(* Logix 5000 project; controller Digital_Interlock_PLC vendor 1 type 14 code 196 rev 37.11; software revision 37.00 *)

TASK HeartbeatTask (periodic, rate 500 ms, priority 6, watchdog 10000 ms) : HeartbeatProgram
TASK MainTask (periodic, rate 5 ms, priority 5, watchdog 500 ms) : MainProgram
TASK ManageOptimizationTask (continuous, watchdog 500 ms) : ManageOptimizationProgram

MODULES
   Local : vendor 1 type 14 code 196 (5069 0, rev 37.11)
      PF1 : vendor 1 type 14 code 107 (Ethernet 10.10.10.48, rev 37.1)
      PR1 : vendor 887 type 12 code 42780 (Ethernet 10.10.10.6, rev 1.37, StandardDataDriven RPI 5 ms)
      ST1 : vendor 887 type 12 code 42780 (Ethernet 10.10.10.59, rev 1.37, StandardDataDriven RPI 5 ms)
END_MODULES

TYPE STR_MajorFault :
STRUCT
   LEN : DINT;
   DATA : SINT[300];
END_STRUCT
END_TYPE

TYPE UDT_Comms :
STRUCT
   PF : UDT_CommsHealth;
   PR : UDT_CommsHealth;
   ST : UDT_CommsHealth;
END_STRUCT
END_TYPE

TYPE UDT_CommsHealth :
STRUCT
   CommsError : BOOL;
   Healthy : BOOL;
   HeartbeatChanged : BOOL;
   Inhibited : BOOL;   // inhibited/uninhibited
   FaultInfo : DINT;
   Heartbeat : DINT;
   Inhibit : DINT;   // 0 to unihibit, 4 to inhibit.
   Instance : DINT;
   ArrivalPeriod_ms : REAL;
   Jitter_ms : REAL;
   LastArrivalPeriod_ms : REAL;
   Latency_ms : REAL;
   LatencyPeak_ms : REAL;
   LatencyAvg_ms : REAL;
   FaultCode : INT;   // 515 (disconnected during use), 516 (disconnected before controller run mode)
   Mode : INT;   // 0 (causes a major fault to be generated if any of the Module object connections fault while the controller is in Run mode) 2 (causes the Module object to enter Inhibited state after shutting down all the connections to the module.)
   Path : SINT[2];
END_STRUCT
END_TYPE

TYPE UDT_FaultRecord :
STRUCT
   TimeLow : DINT;
   TimeHigh : DINT;
   Type : INT;
   Code : INT;
   Info : DINT[11];
END_STRUCT
END_TYPE

TYPE UDT_FromLIC :   // Data that is exchanged with LIC Client
STRUCT
   EnableLineOptimization : BOOL;
   Deadband : DINT;
   FeedInterruptSetting : DINT;
   MaxCommandSpeed : DINT;
   MinCommandSpeed : DINT;
   Proportional : DINT;
   SampleRate : DINT;
   TargetFillPercentage : DINT;
   MachineList : STRING;
END_STRUCT
END_TYPE

TYPE UDT_MachineLFOProperties :   // UDT containing members needed for line flow optimization
STRUCT
   FeedInterruptStatus : BOOL;
   CommandedSpeed : DINT;
   CurrentSpeed : DINT;
   CurrentFillPercent : DINT;
   DeadBand : DINT;
   FeedInterruptSetting : DINT;
   PatternMaxSpeed : DINT;
   PatternMinSpeed : DINT;
   ReferenceSpeed : DINT;
   SpeedCalcRate : DINT;
   TargetFillPercent : DINT;
END_STRUCT
END_TYPE

TYPE UDT_MSG :
STRUCT
   To : DINT[33];
   From : DINT[33];
END_STRUCT
END_TYPE

TYPE UDT_ToLIC :
STRUCT
   FeedInterrupt : BOOL;   // Feed interrupt executed
   FeedInterrupted : BOOL;   // Interrupt completed
   CommsHealthy : BOOL;   // All machines are communicating
   MachinesConnected : BOOL[32];   // Boolean array that contains machine connection status
END_STRUCT
END_TYPE

ADD_ON_INSTRUCTION AOI_Calculate_Latency   (* revision 1.0 *)
VAR_INPUT
   Inp_DeviceHeartbeat : DINT; {required}
   Inp_CurrentTime_us : DINT; {required}
END_VAR
VAR_OUTPUT
   Out_LastTime_ms : DINT; {access Read Only, required}
   Out_HeartbeatChanged : BOOL; {access Read Only, required}
END_VAR
VAR
   CurrentTime_ms : DINT; {access None}
   PreviousTime_ms : DINT; {access None}
   PreviousHeartbeat : DINT; {access None}
   PreviousTime_us : DINT; {access None}
   dt_us : DINT; {access None}
   dt_ms : DINT; {access None}
END_VAR

ROUTINE Logic   (* structured text *)
   (*----------------------------------------------------------
   ROLLOVER-SAFE TIME DELTA
   	Inp_Timestamp_us is a microsecond counter that rolls to
   	zero each period. If the current timestamp is less than
   	the previous one, treat it as a rollover case.
   ----------------------------------------------------------*)
   
   if Inp_CurrentTime_us >= PreviousTime_us then
   	// Normal delta
       dt_us := Inp_CurrentTime_us - PreviousTime_us;
   else
   	// Rollover delta = remaining to modulus + current
   	dt_us := (1000000 - PreviousTime_us) + Inp_CurrentTime_us;
   end_if;
   
   // Convert microseconds to milliseconds for outputs.
   dt_ms := (dt_us) / 1000.0;
   
   
   if Inp_DeviceHeartbeat <> PreviousHeartbeat then
   	Out_HeartbeatChanged := 1;
   	Out_LastTime_ms := dt_ms - PreviousTime_ms;
   	PreviousTime_ms := dt_ms;
   else
   	Out_HeartbeatChanged := 0;
   end_if;
   
   PreviousHeartbeat := Inp_DeviceHeartbeat;
END_ROUTINE
END_ADD_ON_INSTRUCTION

ADD_ON_INSTRUCTION AOI_Detect_Heartbeat   (* revision 1.0 *)
VAR_INPUT
   Inp_Heartbeat : DINT; {required}
   Inp_WatchdogTime_ms : DINT; {visible}
END_VAR
VAR_OUTPUT
   Out_Heartbeat_Changed : BOOL; {access Read Only, visible}
   Out_WD_DN : BOOL; {access Read Only, visible}
   Out_WD_ACC : DINT; {access Read Only, visible}
   Out_WD_EN : BOOL; {access Read Only, visible}
   Out_Heartbeat_Healthy : BOOL; {access Read Only, required}
END_VAR
VAR
   PreviousHeartbeat : DINT; {access None}
   CurrentHeartbeat : DINT; {access None}
   HeartbeatWatchdog : FBD_TIMER; {access None}
END_VAR

ROUTINE Logic   (* structured text *)
   // Update current heartbeat value
   CurrentHeartbeat := Inp_Heartbeat;
   // Monitor changes in heartbeat
   Out_Heartbeat_Changed := (CurrentHeartbeat <> PreviousHeartbeat); //AND (NOT HeartbeatWatchdog.DN);
   
   // Check and set default preset for the watchdog if input preset is invalid (default to 10s)
   TONR(HeartbeatWatchdog);
   if Inp_WatchdogTime_ms <= 10000 then
   	HeartbeatWatchdog.PRE := 10000;
   else
   	HeartbeatWatchdog.PRE := Inp_WatchdogTime_ms;
   end_if;
   
   
   // Enable the watchdog timer if the heartbeat stops changing
   HeartbeatWatchdog.TimerEnable := NOT Out_Heartbeat_Changed;
   
   // Indicate bad health if the watchdog completes and no heartbeat change is detected
   Out_Heartbeat_Healthy := NOT (HeartbeatWatchdog.DN AND NOT Out_Heartbeat_Changed);
   
   // Reset the watchdog if both enabled and heartbeat changes detected
   if HeartbeatWatchdog.TimerEnable AND Out_Heartbeat_Changed then
       HeartbeatWatchdog.Reset := 1;
       HeartbeatWatchdog.TimerEnable := 0;
       HeartbeatWatchdog.Reset := 0;
   end_if;
   
   // Output the watchdog status flags
   Out_WD_DN := HeartbeatWatchdog.DN;
   Out_WD_ACC := HeartbeatWatchdog.ACC;
   Out_WD_EN := HeartbeatWatchdog.EN;
   
   // Store the current heartbeat for the next cycle
   PreviousHeartbeat := CurrentHeartbeat;
END_ROUTINE
END_ADD_ON_INSTRUCTION

ADD_ON_INSTRUCTION AOI_Monitor_Comms   (* revision 1.0 *)
// Latency-monitoring AOI tracks:
// Last heartbeat value
// Timestamp of last sample
// Latency (current, average, peak)
// Jitter (simple absolute-difference model)
VAR_INPUT
   Inp_Heartbeat : DINT; {required}   // heartbeat counter received from remote device
   Inp_Timestamp_us : DINT; {required}   // wall-clock microseconds from GSV(WallClockTime)
   Inp_MaxSameScans : DINT; {required}
   Inp_Rollover_us : DINT; {required}
   Inp_SmoothingFactor : REAL; {required}
   Inp_Reset : BOOL; {required}
END_VAR
VAR_OUTPUT
   Out_Latency_ms : REAL; {required}
   Out_LatencyAvg_ms : REAL; {access Read Only, required}
   Out_LatencyPeak_ms : REAL; {access Read Only, required}
   Out_Jitter_ms : REAL; {access Read Only, required}
   Out_Fresh : BOOL; {access Read Only, required}
   Out_HeartbeatOK : BOOL; {access Read Only, required}
END_VAR
VAR
   EMA : REAL; {access None}   // exponential smoothing accumulator
   FirstScan : BOOL; {access None}
   PreviousTime_us : DINT; {access None}
   PreviousHeartbeat : DINT; {access None}
   dt_us : DINT; {access None}
   dt_ms : REAL; {access None}
   SameValue : DINT; {access None}
   HeartbeatTimer : FBD_TIMER; {access None}
   EMA_prev : REAL; {access None}
   alpha : REAL; {access None}
   modulus : DINT; {access None}
END_VAR

ROUTINE Logic   (* structured text *)
// Latency-monitoring AOI
// It tracks:
// Last heartbeat value
// Timestamp of last sample
// Latency (current, average, peak)
// Jitter (simple absolute-difference model)
   (*
   |=================================================================|
   |						AOI_Comms_Monitor						  |
   |_________________________________________________________________|
   | Purpose:														  |
   | 	Measure time between successive remote heartbeats to estimate |
   |	comms latency, while handling microsecond timestamp rollover. |
   |																  |
   | Outputs are in milliseconds.									  |
   |_________________________________________________________________|
   *)
   
   (*--------------------------------------------------------------
   DISABLE / RESET BEHAVIOR
   	When disabled or reset, clear diagnostics and re-arm the
   	first-scan latch so the next enable reinitializes state.
   --------------------------------------------------------------*)
   
   if (NOT EnableIn) OR Inp_Reset then
   	FirstScan := 1;							// Force re-init on next enabled scan
   	PreviousTime_us := Inp_Timestamp_us;	// Seed previous timestamp to current
   	PreviousHeartbeat := Inp_Heartbeat;		// Seed previous heartbeat to current
   	EMA := 0;								// Clear exponential moving average accumulator
   	EMA_prev := 0;
   	SameValue := 0;
   
   	// Clear all status/diagnostics while disabled
   	Out_Fresh := 0;
   	Out_Latency_ms := 0;
   	Out_LatencyAvg_ms := 0;
   	Out_LatencyPeak_ms := 0;
   	Out_Jitter_ms := 0;
   	Out_HeartbeatOK := 0;
   end_if;
   
   (*--------------------------------------------------------------
   FIRST SAMPLE INITIALIZATION
   	On the first enabled scan, capture the baseline heartbeat
   	and timestamp so the next fresh value can compute a delta.
   --------------------------------------------------------------*)
   if FirstScan then
   	FirstScan := 0;							// Clear first-scan latch
   	PreviousHeartbeat := Inp_Heartbeat;		// Store current HB as baseline
   	PreviousTime_us := Inp_Timestamp_us;	// Store current timestamp as baseline
   
   	EMA := 0.0;								// Reset filter state
   	EMA_prev := 0.0;
   	SameValue := 0;
   
   	Out_HeartbeatOK := 1;					// Consider OK after initialization
   	Out_Fresh := 0;
   	Out_Latency_ms := 0.0;
   	Out_LatencyAvg_ms := 0.0;
   	Out_LatencyPeak_ms := 0.0;
   	Out_Jitter_ms := 0.0;
   end_if;
   
   
   (*--------------------------------------------------------------
   INPUT VALIDATION
   	Ensure smoothing factor is bounded between 0.0 and 1.0.
   	A heartbeat is considered "fresh" when its counter changes.
   --------------------------------------------------------------*)
   if Inp_SmoothingFactor < 0.0 then
   	Inp_SmoothingFactor := 0.0;
   end_if;
   
   if Inp_SmoothingFactor > 1.0 then
   	Inp_SmoothingFactor := 1.0;
   end_if;
   
   IF Inp_Rollover_us = 0 then
   	// Invalid modulus: mark unhealthy and bail (why: cannot compute deltas)
   	Out_Fresh := 0;
   	Out_HeartbeatOK := 0;
   end_if;
   
   
   (*--------------------------------------------------------------
   DETECT NEW HEARTBEAT
   	A heartbeat is considered "fresh" when its counter changes.
   --------------------------------------------------------------*)
   Out_Fresh := (Inp_Heartbeat <> PreviousHeartbeat);
   
   if Out_Fresh then
   	(*----------------------------------------------------------
   	ROLLOVER-SAFE TIME DELTA
   		Inp_Timestamp_us is a microsecond counter that rolls to
   		zero each period. If the current timestamp is less than
   		the previous one, treat it as a rollover case.
   	----------------------------------------------------------*)
   	if Inp_Timestamp_us >= PreviousTime_us then
   	    dt_us := Inp_Timestamp_us - PreviousTime_us;						// Normal delta
   	else
   		dt_us := (Inp_Rollover_us - PreviousTime_us) + Inp_Timestamp_us;	// Rollover delta = remaining to modulus + current
   	end_if;
   
   	dt_ms := (dt_us) / 1000.0;			// Convert microseconds to milliseconds for outputs.
   
   	Out_Latency_ms := dt_ms;			// Latency for this heartbeat interval
   
   	if dt_ms > Out_LatencyPeak_ms then
   		Out_LatencyPeak_ms := dt_ms;	// Track worst-case latency
   	end_if;
   
   	(*----------------------------------------------------------
   	SMOOTHED AVERAGE (EMA)
   		EMA is a low-pass filter:
   			EMA := (1 - alpha) * EMA + alpha * sample
   		Here, alpha is provided as Inp_SmoothingFactor.
   	----------------------------------------------------------*)
   
   	EMA := (1-Inp_SmoothingFactor) * EMA + Inp_SmoothingFactor * dt_ms;
   
   	Out_LatencyAvg_ms := EMA;
   
   	(*----------------------------------------------------------
   	JITTER ESTIMATE
   		Jitter is modeled as the absolute deviation of the
   		latest sample from the smoothed average.
   	----------------------------------------------------------*)
   	Out_Jitter_ms := ABS(dt_ms - EMA);
   
   	(*----------------------------------------------------------
   	UPDATE HISTORY
   		Persist current values for the next fresh heartbeat
   		comparison and mark comms as healthy.
   	----------------------------------------------------------*)
   	PreviousHeartbeat := Inp_Heartbeat;
   	PreviousTime_us := Inp_Timestamp_us;
   	SameValue := 0;
   	Out_HeartbeatOK := 1;
   
   else
   	// Heartbeat did not change this scan; track consecutive repeats
   	if SameValue < Inp_MaxSameScans then
   		SameValue := SameValue + 1;
   	end_if;
   
   	// After N identical scans, consider comms unhealthy
   	if (SameValue >= Inp_MaxSameScans) then
   		Out_HeartbeatOK := 0;
   	end_if;
   end_if;
END_ROUTINE
END_ADD_ON_INSTRUCTION

ADD_ON_INSTRUCTION AOI_Optimize_Flow   (* revision 1.0 *)
// Line Speed Adjustment
VAR_INPUT
   Inp_CurrentSpeed : DINT; {required}   // Current speed of the target machine (KPM)
   Inp_ReferenceSpeed : DINT; {required}   // Reference speed of the downstream machine (KPM)
   Inp_CurrentFillPercent : DINT; {required}
   Inp_TargetFillPercent : DINT; {required}   // Target Fill Percentage, the desired fill percentage to achieve by adjusting speeds (%)
   Inp_MaxSpeed : DINT; {required}   // Maximum speed of job (KPM)
   Inp_MinSpeed : DINT; {required}   // Minimum speed of target machine (KPM)
   Inp_FeedInterruptSetting : DINT; {required}   // Value set by LIC Client user interface
   Inp_SpeedCalcRate : DINT; {required}   // Rate of speed calculations
END_VAR
VAR_OUTPUT
   Out_CommandSpeed : DINT; {required}
   Out_FeedInterrupt : BOOL; {required}   // Value set to TRUE, when the Reference Fill % is equal to or greater than the Feed Interrupt Setting LIC Client user input).
END_VAR
VAR
   SpeedCalcTimer : TIMER;
   ProportionalGain : DINT;   // Proportial multiple to adjust aggressiveness of changes to speed commands, limited to [0.5 - 1.2]
   DeadBand : DINT;   // Value that represents the amount of percentage points from target fill percentage that the current fill percentage must be before calculating command speed
   LowerDeadBand : DINT;
   UpperDeadBand : DINT;
END_VAR

ROUTINE Logic   (* ladder *)
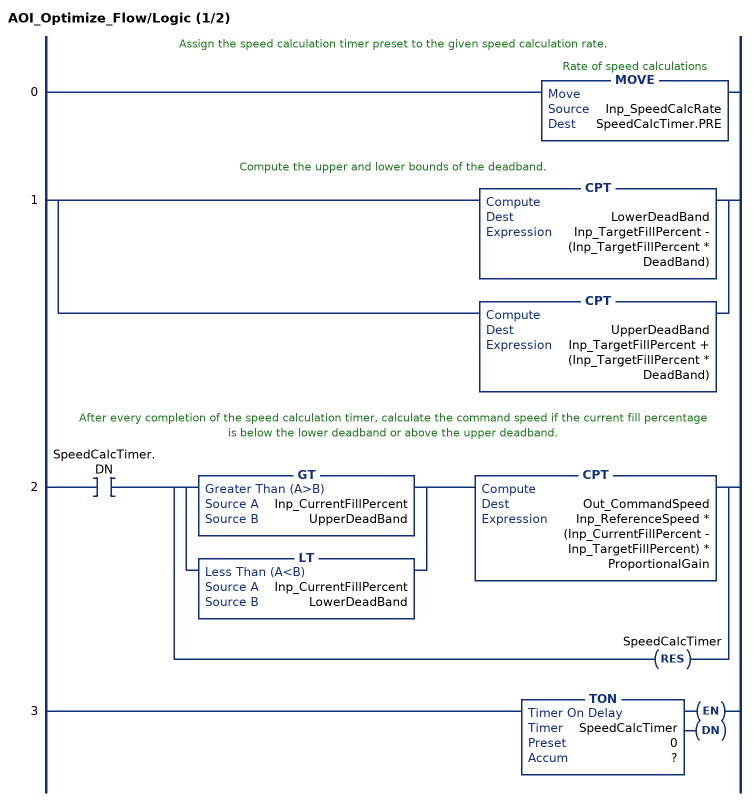
   // Assign the speed calculation timer preset to the given speed calculation rate.
   0: MOVE(Inp_SpeedCalcRate,SpeedCalcTimer.PRE);
   // Compute the upper and lower bounds of the deadband.
   1: [CPT(LowerDeadBand,Inp_TargetFillPercent - (Inp_TargetFillPercent * DeadBand)) ,CPT(UpperDeadBand,Inp_TargetFillPercent + (Inp_TargetFillPercent * DeadBand)) ];
   // After every completion of the speed calculation timer, calculate the command speed if the current fill percentage is below the lower deadband or above the upper deadband.
   2: XIC(SpeedCalcTimer.DN)[[GT(Inp_CurrentFillPercent,UpperDeadBand) ,LT(Inp_CurrentFillPercent,LowerDeadBand) ] CPT(Out_CommandSpeed,Inp_ReferenceSpeed * (Inp_CurrentFillPercent - Inp_TargetFillPercent) * ProportionalGain) ,RES(SpeedCalcTimer) ];
   3: TON(SpeedCalcTimer,?,?);
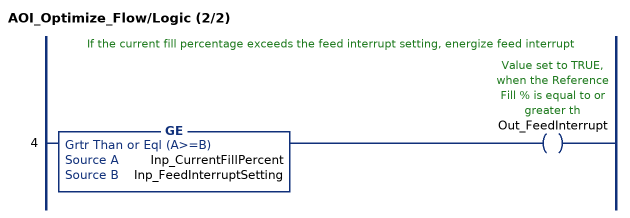
   // If the current fill percentage exceeds the feed interrupt setting, energize feed interrupt
   4: GE(Inp_CurrentFillPercent,Inp_FeedInterruptSetting)OTE(Out_FeedInterrupt);
END_ROUTINE
END_ADD_ON_INSTRUCTION

VAR_GLOBAL   (* controller tags *)
   _DEBUG : BOOL;
   AlwaysTrue : BOOL := 1; {constant}
   CommsStatus : DINT := 7;
        .0   // Bit for PREFEEDER Comms Status
        .3   // Bit for LIC Comms Status
        .2   // Bit for STACKER Comms Status
        .1   // Bit for PRESS Comms Status
   CurrentTime : DINT[7] := ([0] := 2026, [1] := 2, [2] := 23, [3] := 14, [4] := 10, [5] := 41, [6] := 704831);
   EnableLineOptimization : BOOL;
   FromPrefeeder : DINT[33] := ([0] := 264, [3] := 734);   // DINTs used: 0-2
        [0].8   // (Pre-Feeder -> Press) FromPrefeeder.MachineOpenCloseDisable
        [0].11   // (Pre-Feeder -> Press) FromPrefeeder.ReadyToRaise
        [0].1   // (Pre-Feeder -> Press) FromPrefeeder.AuxTamperAirLeft
        [0].10   // (Pre-Feeder -> Press) FromPrefeeder.ReadyForSetup
        [0].7   // (Pre-Feeder -> Press) FromPrefeeder.FeedBoardOk
        [2]   // (Pre-Feeder -> Press) FromPrefeeder.PatternMaxSpeed
        [0].5   // (Pre-Feeder -> Press) FromPrefeeder.EstopFeedbackChannel1
        [0].6   // (Pre-Feeder -> Press) FromPrefeeder.EstopFeedbackChannel2
        [0].2   // (Pre-Feeder -> Press) FromPrefeeder.BackstopInhibit
        [0].4   // (Pre-Feeder -> Press) FromPrefeeder.ExtendoUpDown
        [0].18   // Spare
        [4]   // (Pre-Feeder -> Press) FromPrefeeder.Spare1
        [1]   // (Pre-Feeder -> Press) FromPrefeeder.CurrentSpeed
        [3]   // (Pre-Feeder -> Press) FromPrefeeder.Heartbeat
        [5]   // (Pre-Feeder -> Press) FromPrefeeder.Spare2
        [0].19   // Spare
        [0].20   // Spare
        [0].12   // (Pre-Feeder -> Press) FromPrefeeder.RunEmpty
        [0].21   // Spare
        [0].22   // Spare
        [0].23   // Spare
        [0].24   // Spare
        [0]   // Bits used: 0-17
        [0].9   // (Pre-Feeder -> Press) FromPrefeeder.OpenMachineOk
        [0].16   // (Pre-Feeder -> Press) FromPrefeeder.Empty
        [0].17   // (Pre-Feeder -> Press) FromPrefeeder.Spare
        [0].0   // (Pre-Feeder -> Press) FromPrefeeder.AuxTamperAirRight
        [10]   // Spare
        [11]   // Spare
        [12]   // Spare
        [13]   // Spare
        [14]   // Spare
        [15]   // Spare
        [16]   // Spare
        [17]   // Spare
        [18]   // Spare
        [19]   // Spare
        [20]   // Spare
        [21]   // Spare
        [22]   // Spare
        [23]   // Spare
        [24]   // Spare
        [25]   // Spare
        [26]   // Spare
        [27]   // Spare
        [28]   // Spare
        [0].13   // (Pre-Feeder -> Floor Conv) FromPrefeeder.RunForward
        [0].14   // (Pre-Feeder -> Floor Conv) FromPrefeeder.RunReverse
        [0].15   // (Pre-Feeder -> Press) FromPrefeeder.TamperInterrupt
        [0].3   // (Pre-Feeder -> Floor Conv) FromPrefeeder.CallForStack
        [0].25   // Spare
        [0].26   // Spare
        [0].27   // Spare
        [0].28   // Spare
        [0].29   // Spare
        [0].30   // Spare
        [0].31   // Spare
        [29]   // Spare
        [30]   // Spare
        [31]   // Spare
        [32]   // Spare
        [6]   // Spare
        [7]   // Spare
        [8]   // Spare
        [9]   // Spare
   FromPrefeeder_Copied : REAL[20];
   FromPress : DINT[33] := ([0] := 60635, [1] := 125, [2] := 75, [3] := 16, [4] := 888, [5] := 1143336141, [7] := 1153686979, [8] := 1153638072, [9] := 1153709834, [14] := 1146431734, [15] := -1098572104);
   FromPress_Copied : REAL[20];
   FromStacker : DINT[33];   // DINTS used: 0-22
        [4].7   // (Stacker -> Press) fromStacker.DieCutter.blnRegisterStopAdjustRq
        [4].3   // (Stacker -> Press) fromStacker.FeedInterruptStatus
        [4].6   // (Stacker -> Press) fromStacker.DieCutter.blnRegisterAdjustRq
        [4].9   // (Stacker -> Press) fromStacker.DieCutter.blnSidewaysStopAdjustRq
        [5].0   // (Stacker -> Press) fromStacker.PrintStation[7].blnRegisterStopAdjustRq
        [4].4   // (Stacker -> Press) fromStacker.DieCutter.blnFast
        [10]   // (Stacker -> Press) fromStacker.PrintStation[3].fltDesiredRegisterAdjust
        [4].26   // (Stacker -> Press) fromStacker.PrintStation[1].blnRegisterStopAdjustRq
        [4].8   // (Stacker -> Press) fromStacker.DieCutter.blnSidewaysAdjustRq
        [7]   // (Stacker -> Press) fromStacker.DieCutter.fltDesiredRegisterAdjust
        [15]   // (Stacker -> Press) fromStacker.DieCutter.fltDesiredSidewaysAdjust
        [4].10   // (Stacker -> Press) fromStacker.DieCutter.blnSpeedChangeRq
        [5].1   // (Stacker -> Press) fromStacker.PrintStation[1].blnSidewaysStopAdjustRq
        [4].12   // (Stacker -> Press) fromStacker.PrintStation[1].blnRegisterAdjustRq
        [5].2   // (Stacker -> Press) fromStacker.PrintStation[2].blnSidewaysStopAdjustRq
        [4].11   // (Stacker -> Press) fromStacker.DieCutter.blnSpeedChangeStopRq
        [5].3   // (Stacker -> Press) fromStacker.PrintStation[3].blnSidewaysStopAdjustRq
        [11]   // (Stacker -> Press) fromStacker.PrintStation[4].fltDesiredRegisterAdjust
        [8]   // (Stacker -> Press) fromStacker.PrintStation[1].fltDesiredRegisterAdjust
        [5].4   // (Stacker -> Press) fromStacker.PrintStation[4].blnSidewaysStopAdjustRq
        [9]   // (Stacker -> Press) fromStacker.PrintStation[2].fltDesiredRegisterAdjust
        [5].5   // (Stacker -> Press) fromStacker.PrintStation[5].blnSidewaysStopAdjustRq
        [4].13   // (Stacker -> Press) fromStacker.PrintStation[2].blnRegisterAdjustRq
        [5].6   // (Stacker -> Press) fromStacker.PrintStation[6].blnSidewaysStopAdjustRq
        [6]   // (Stacker -> Press) fromStacker.DieCutter.uiDesiredSpeedKpm
        [4].14   // (Stacker -> Press) fromStacker.PrintStation[3].blnRegisterAdjustRq
        [4].15   // (Stacker -> Press) fromStacker.PrintStation[4].blnRegisterAdjustRq
        [4].16   // (Stacker -> Press) fromStacker.PrintStation[5].blnRegisterAdjustRq
        [12]   // (Stacker -> Press) fromStacker.PrintStation[5].fltDesiredRegisterAdjust
        [13]   // (Stacker -> Press) fromStacker.PrintStation[6].fltDesiredRegisterAdjust
        [14]   // (Stacker -> Press) fromStacker.PrintStation[7].fltDesiredRegisterAdjust
        [16]   // (Stacker -> Press) fromStacker.PrintStation[1].fltDesiredSidewaysAdjust
        [17]   // (Stacker -> Press) fromStacker.PrintStation[2].fltDesiredSidewaysAdjust
        [18]   // (Stacker -> Press) fromStacker.PrintStation[3].fltDesiredSidewaysAdjust
        [19]   // (Stacker -> Press) fromStacker.PrintStation[4].fltDesiredSidewaysAdjust
        [20]   // (Stacker -> Press) fromStacker.PrintStation[5].fltDesiredSidewaysAdjust
        [21]   // (Stacker -> Press) fromStacker.PrintStation[6].fltDesiredSidewaysAdjust
        [22]   // (Stacker -> Press) fromStacker.PrintStation[7].fltDesiredSidewaysAdjust
        [5].7   // (Stacker -> Press) fromStacker.PrintStation[7].blnSidewaysStopAdjustRq
        [4].27   // (Stacker -> Press) fromStacker.PrintStation[2].blnRegisterStopAdjustRq
        [4].17   // (Stacker -> Press) fromStacker.PrintStation[6].blnRegisterAdjustRq
        [4].28   // (Stacker -> Press) fromStacker.PrintStation[3].blnRegisterStopAdjustRq
        [4].18   // (Stacker -> Press) fromStacker.PrintStation[7].blnRegisterAdjustRq
        [4].19   // (Stacker -> Press) fromStacker.PrintStation[1].blnSidewaysAdjustRq
        [4].5   // (Stacker -> Press) fromStacker.DieCutter.blnSlow
        [4].2   // (Stacker -> Press) fromStacker.RolledOutStatus
        [4].0   // (Stacker -> Press) fromStacker.RunPermissive
        [4].29   // (Stacker -> Press) fromStacker.PrintStation[4].blnRegisterStopAdjustRq
        [4].30   // (Stacker -> Press) fromStacker.PrintStation[5].blnRegisterStopAdjustRq
        [4].31   // (Stacker -> Press) fromStacker.PrintStation[6].blnRegisterStopAdjustRq
        [4].20   // (Stacker -> Press) fromStacker.PrintStation[2].blnSidewaysAdjustRq
        [4].21   // (Stacker -> Press) fromStacker.PrintStation[3].blnSidewaysAdjustRq
        [2]   // (Stacker -> Press) fromStacker.PatternMaxSpeed
        [4].1   // (Stacker -> Press) fromStacker.FeedRestart
        [0]   // (Stacker -> Press) fromStacker.Heartbeat
        [3]   // (Stacker -> Press) fromStacker.FillPercentage
        [5]   // Bits used: 0-7
        [1]   // (Stacker -> Press) fromStacker.CurrentSpeed
        [4].22   // (Stacker -> Press) fromStacker.PrintStation[4].blnSidewaysAdjustRq
        [4]   // Bits used: 0-31
        [4].23   // (Stacker -> Press) fromStacker.PrintStation[5].blnSidewaysAdjustRq
        [4].24   // (Stacker -> Press) fromStacker.PrintStation[6].blnSidewaysAdjustRq
        [4].25   // (Stacker -> Press) fromStacker.PrintStation[7].blnSidewaysAdjustRq
        [23]   // Spare
        [24]   // Spare
        [25]   // Spare
        [26]   // Spare
        [27]   // Spare
        [28]   // Spare
        [29]   // Spare
        [30]   // Spare
        [31]   // Spare
        [32]   // Spare
   FromStacker_Copied : REAL[20];
   HeartbeatCounter : INT := 832;
   PF_Comms : UDT_CommsHealth;
        .CommsError   // Prefeeder comms error
   PR_Comms : UDT_CommsHealth;
        .CommsError   // Press comms error
   PrefeederData : UDT_MSG := (To[8] := 727, To[9] := 7, From[0] := 264, From[3] := 727);
   PrefeederLFO : UDT_MachineLFOProperties;
   PrefeederLFO_AOI : AOI_Optimize_Flow;
   PrefeederMSG : MESSAGE;
        MessageParameters(ServiceCode := 16#004d, LocalElement := PrefeederData.To[0], ...)
   PressLatency_AOI : AOI_Calculate_Latency;
   PressLFO : UDT_MachineLFOProperties;
   PressLFO_AOI : AOI_Optimize_Flow;
   ST_Comms : UDT_CommsHealth;
        .CommsError   // Stacker comms error
   StackerLFO : UDT_MachineLFOProperties;
   StackerLFO_AOI : AOI_Optimize_Flow;
   ToPrefeeder2 : DINT[33];   // DINTs used: 0-11
        [4]   // (Press -> Pre-Feeder) ToPrefeeder.HopperHeightSetpoint
        [0].10   // ToPrefeeder.ShuttleCarAtPrefeeder (Floor Conv -> Prefeeder)
        [0].9   // ToPrefeeder.StackReadyInFeed (Floor Conv -> Prefeeder)
        [0].4   // ToPrefeeder.LastStack (Floor Conv -> Prefeeder)
        [7]   // (Press -> Pre-Feeder) ToPrefeeder.LinearSpeedActual
        [0].3   // ToPrefeeder.ExtendoFollowBackstopDown (Press -> Pre-Feeder)
        [0].2   // ToPrefeeder.ExtendoFollowBackstopUp (Press -> Pre-Feeder)
        [0].8   // ToPrefeeder.RequestOpen (Press -> Pre-Feeder)
        [5]   // (Press -> Pre-Feeder) ToPrefeeder.HopperHeightMin
        [9]   // (Interlock -> Pre-Feeder) ToPrefeeder.CommsStatus
        [27]   // Spare
        [28]   // Spare
        [29]   // Spare
        [30]   // Spare
        [0].25   // Spare
        [0].6   // ToPrefeeder.MachineInFeedMode (Press -> Pre-Feeder)
        [0].26   // Spare
        [0].27   // Spare
        [31]   // Spare
        [0].28   // Spare
        [0].29   // Spare
        [0].30   // Spare
        [0].31   // Spare
        [0].7   // ToPrefeeder.MachineRunning (Press -> Pre-Feeder)
        [0].5   // ToPrefeeder.LoadHopper (Press -> Pre-Feeder)
        [1]   // (Press -> Pre-Feeder) ToPrefeeder.CommandedSpeed
        [2]   // (Press -> Pre-Feeder) ToPrefeeder.BoardCaliper
        [8]   // Prefeeder[8] (ToPrefeeder.Heartbeat)
        [10]   // (Press -> Pre-Feeder) ToPrefeeder.Spare1
        [11]   // (Press -> Pre-Feeder) ToPrefeeder.Spare2
        [0].1   // ToPrefeeder.ConvRunning (Floor Conv -> Prefeeder)
        [0]   // Bits used: 0-10
        [0].0   // ToPrefeeder.ClosedLocked (Press -> Pre-Feeder)
        [3]   // (Press -> Pre-Feeder) ToPrefeeder.FeedHopperHeight
        [6]   // (Press -> Pre-Feeder) ToPrefeeder.LinearSpeedSetpoint
        [0].11   // Spare
        [0].12   // Spare
        [0].13   // Spare
        [0].14   // Spare
        [0].15   // Spare
        [0].16   // Spare
        [0].17   // Spare
        [12]   // Spare
        [13]   // Spare
        [14]   // Spare
        [15]   // Spare
        [16]   // Spare
        [17]   // Spare
        [18]   // Spare
        [19]   // Spare
        [20]   // Spare
        [21]   // Spare
        [22]   // Spare
        [23]   // Spare
        [24]   // Spare
        [25]   // Spare
        [26]   // Spare
        [0].18   // Spare
        [0].19   // Spare
        [0].20   // Spare
        [0].21   // Spare
        [0].22   // Spare
        [0].23   // Spare
        [0].24   // Spare
   ToPress : DINT[40];   // DINTs used: 0-32
        [10].6   // (Stacker -> Press) fromStacker.DieCutter.blnRegisterAdjustRq
        [10].8   // (Stacker -> Press) fromStacker.DieCutter.blnSidewaysAdjustRq
        [0].1   // (Pre-Feeder -> Press) FromPrefeeder.AuxTamperAirLeft
        [12]   // (Stacker -> Press) fromStacker.DieCutter.uiDesiredSpeedKpm
        [0].11   // (Pre-Feeder -> Press) FromPrefeeder.ReadyToRaise
        [0].5   // (Pre-Feeder -> Press) FromPrefeeder.EstopFeedbackChannel1
        [0].10   // (Pre-Feeder -> Press) FromPrefeeder.ReadyForSetup
        [10].11   // (Stacker -> Press) fromStacker.DieCutter.blnSpeedChangeStopRq
        [10].26   // (Stacker -> Press) fromStacker.PrintStation[1].blnRegisterStopAdjustRq
        [10].7   // (Stacker -> Press) fromStacker.DieCutter.blnRegisterStopAdjustRq
        [10].9   // (Stacker -> Press) fromStacker.DieCutter.blnSidewaysStopAdjustRq
        [10].27   // (Stacker -> Press) fromStacker.PrintStation[2].blnRegisterStopAdjustRq
        [10].28   // (Stacker -> Press) fromStacker.PrintStation[3].blnRegisterStopAdjustRq
        [0].17   // (Pre-Feeder -> Press) FromPrefeeder.FeedInterrupt
        [10].4   // (Stacker -> Press) fromStacker.DieCutter.blnFast
        [10].29   // (Stacker -> Press) fromStacker.PrintStation[4].blnRegisterStopAdjustRq
        [10].3   // (Stacker -> Press) FromStacker.FeedInterruptStatus
        [10].10   // (Stacker -> Press) fromStacker.DieCutter.blnSpeedChangeRq
        [32].0   // (Interlock -> Prefeeder) FromInterlock.PrefeederCommsStatus
        [10].5   // (Stacker -> Press) fromStacker.DieCutter.blnSlow
        [10].30   // (Stacker -> Press) fromStacker.PrintStation[5].blnRegisterStopAdjustRq
        [10].31   // (Stacker -> Press) fromStacker.PrintStation[6].blnRegisterStopAdjustRq
        [0].8   // (Pre-Feeder -> Press) FromPrefeeder.MachineOpenCloseDisable
        [0].6   // (Pre-Feeder -> Press) FromPrefeeder.EstopFeedbackChannel2
        [13]   // (Stacker -> Press) fromStacker.DieCutter.fltDesiredRegisterAdjust
        [21]   // (Stacker -> Press) fromStacker.DieCutter.fltDesiredSidewaysAdjust
        [0].2   // (Pre-Feeder -> Press) FromPrefeeder.BackstopInhibit
        [0].7   // (Pre-Feeder -> Press) FromPrefeeder.FeedBoardOk
        [2]   // (Pre-Feeder -> Press) FromPrefeeder.PatternMaxSpeed
        [31]   // (Interlock -> Press) FromInterlock.CommandedSpeed
        [14]   // (Stacker -> Press) fromStacker.PrintStation[1].fltDesiredRegisterAdjust
        [15]   // (Stacker -> Press) fromStacker.PrintStation[2].fltDesiredRegisterAdjust
        [32].2   // (Interlock -> Stacker) FromInterlock.StackerCommsStatus
        [16]   // (Stacker -> Press) fromStacker.PrintStation[3].fltDesiredRegisterAdjust
        [10].12   // (Stacker -> Press) fromStacker.PrintStation[1].blnRegisterAdjustRq
        [0].0   // (Pre-Feeder -> Press) FromPrefeeder.AuxTamperAirRight
        [17]   // (Stacker -> Press) fromStacker.PrintStation[4].fltDesiredRegisterAdjust
        [18]   // (Stacker -> Press) fromStacker.PrintStation[5].fltDesiredRegisterAdjust
        [10].13   // (Stacker -> Press) fromStacker.PrintStation[2].blnRegisterAdjustRq
        [19]   // (Stacker -> Press) fromStacker.PrintStation[6].fltDesiredRegisterAdjust
        [11].0   // (Stacker -> Press) fromStacker.PrintStation[7].blnRegisterStopAdjustRq
        [20]   // (Stacker -> Press) fromStacker.PrintStation[7].fltDesiredRegisterAdjust
        [22]   // (Stacker -> Press) fromStacker.PrintStation[1].fltDesiredSidewaysAdjust
        [0].4   // (Pre-Feeder -> Press) FromPrefeeder.ExtendoUpDown
        [10].14   // (Stacker -> Press) fromStacker.PrintStation[3].blnRegisterAdjustRq
        [4]   // (Pre-Feeder -> Press) FromPrefeeder.Spare1
        [0].9   // (Pre-Feeder -> Press) FromPrefeeder.OpenMachineOk
        [5]   // (Pre-Feeder -> Press) FromPrefeeder.Spare2
        [11].1   // (Stacker -> Press) fromStacker.PrintStation[1].blnSidewaysStopAdjustRq
        [10].2   // (Stacker -> Press) FromStacker.RolledOutStatus
        [11].2   // (Stacker -> Press) fromStacker.PrintStation[2].blnSidewaysStopAdjustRq
        [11].3   // (Stacker -> Press) fromStacker.PrintStation[3].blnSidewaysStopAdjustRq
        [0].12   // (Pre-Feeder -> Press) FromPrefeeder.RunEmpty
        [32].3   // Spare
        [0].16   // (Pre-Feeder -> Press) FromPrefeeder.Empty
        [32].4   // Spare
        [32].5   // Spare
        [10].1   // (Stacker -> Press) FromStacker.FeedRestart
        [11]   // Bits used: 0-7
        [3]   // (Pre-Feeder -> Press) FromPrefeeder.Heartbeat
        [10]   // Bits uses: 0-31
        [32].6   // Spare
        [32].7   // Spare
        [32].8   // Spare
        [32].9   // Spare
        [32].10   // Spare
        [32]   // Bits used: 0-2
        [32].11   // Spare
        [9]   // (Stacker -> Press) FromStacker.FillPercentage
        [1]   // (Pre-Feeder -> Press) FromPrefeeder.CurrentSpeed
        [10].15   // (Stacker -> Press) fromStacker.PrintStation[4].blnRegisterAdjustRq
        [10].0   // (Stacker -> Press) FromStacker.RunPermissive
        [7]   // (Stacker -> Press) FromStacker.CurrentSpeed
        [11].4   // (Stacker -> Press) fromStacker.PrintStation[4].blnSidewaysStopAdjustRq
        [8]   // (Stacker -> Press) FromStacker.PatternMaxSpeed
        [11].5   // (Stacker -> Press) fromStacker.PrintStation[5].blnSidewaysStopAdjustRq
        [32].12   // Spare
        [29]   // (Stacker -> Press) fromStacker.Spare1
        [10].16   // (Stacker -> Press) fromStacker.PrintStation[5].blnRegisterAdjustRq
        [30]   // (Stacker -> Press) fromStacker.Spare2
        [6]   // (Stacker -> Press) FromStacker.Heartbeat
        [11].6   // (Stacker -> Press) fromStacker.PrintStation[6].blnSidewaysStopAdjustRq
        [0]   // Bits used: 0-18
        [0].13   // (Pre-Feeder -> Floor Conv) FromPrefeeder.RunForward
        [0].14   // (Pre-Feeder -> Floor Conv) FromPrefeeder.RunReverse
        [0].15   // (Pre-Feeder -> Press) FromPrefeeder.TamperInterrupt
        [0].3   // (Pre-Feeder -> Floor Conv) FromPrefeeder.CallForStack
        [32].1   // (Interlock -> Press) FromInterlock.PressCommsStatus
        [0].18   // (Pre-Feeder -> Press) FromPrefeeder.Spare
        [10].17   // (Stacker -> Press) fromStacker.PrintStation[6].blnRegisterAdjustRq
        [10].18   // (Stacker -> Press) fromStacker.PrintStation[7].blnRegisterAdjustRq
        [10].19   // (Stacker -> Press) fromStacker.PrintStation[1].blnSidewaysAdjustRq
        [10].20   // (Stacker -> Press) fromStacker.PrintStation[2].blnSidewaysAdjustRq
        [10].21   // (Stacker -> Press) fromStacker.PrintStation[3].blnSidewaysAdjustRq
        [10].22   // (Stacker -> Press) fromStacker.PrintStation[4].blnSidewaysAdjustRq
        [10].23   // (Stacker -> Press) fromStacker.PrintStation[5].blnSidewaysAdjustRq
        [10].24   // (Stacker -> Press) fromStacker.PrintStation[6].blnSidewaysAdjustRq
        [10].25   // (Stacker -> Press) fromStacker.PrintStation[7].blnSidewaysAdjustRq
        [11].7   // (Stacker -> Press) fromStacker.PrintStation[7].blnSidewaysStopAdjustRq
        [23]   // (Stacker -> Press) fromStacker.PrintStation[2].fltDesiredSidewaysAdjust
        [24]   // (Stacker -> Press) fromStacker.PrintStation[3].fltDesiredSidewaysAdjust
        [25]   // (Stacker -> Press) fromStacker.PrintStation[4].fltDesiredSidewaysAdjust
        [26]   // (Stacker -> Press) fromStacker.PrintStation[5].fltDesiredSidewaysAdjust
        [27]   // (Stacker -> Press) fromStacker.PrintStation[6].fltDesiredSidewaysAdjust
        [28]   // (Stacker -> Press) fromStacker.PrintStation[7].fltDesiredSidewaysAdjust
        [32].13   // Spare
        [32].14   // Spare
        [32].15   // Spare
        [32].16   // Spare
        [32].17   // Spare
        [32].18   // Spare
        [32].19   // Spare
        [32].20   // Spare
        [32].21   // Spare
        [32].22   // Spare
        [32].23   // Spare
        [32].24   // Spare
        [32].25   // Spare
        [32].26   // Spare
        [32].27   // Spare
        [32].28   // Spare
        [32].29   // Spare
        [32].30   // Spare
        [32].31   // Spare
   ToStacker : DINT[33] := ([0] := 60635, [1] := 125, [2] := 75, [3] := 16, [4] := 888, [5] := 1143336141, [7] := 1153686979, [8] := 1153638072, [9] := 1153709834, [14] := 1146431734, [15] := -1098572104);   // DINTS used: 0-23
        [3].15   // (Press -> Stacker) toStacker.PrintStation[1].blnSideWaysActive
        [3].16   // (Press -> Stacker) toStacker.PrintStation[2].blnSideWaysActive
        [3].22   // (LIC -> Stacker) toStacker.DownstreamReady(StraightThru)
        [3].5   // (Press -> Stacker) toStacker.DieCutter.blnRegistrationActive
        [3].8   // (Press -> Stacker) toStacker.PrintStation[1].blnRegistrationActive
        [5]   // (Press -> Stacker) toStacker.DieCutter.fltActualRegisterPosition
        [3].9   // (Press -> Stacker) toStacker.PrintStation[2].blnRegistrationActive
        [3].6   // (Press -> Stacker) toStacker.DieCutter.blnSidewaysAcitve
        [6]   // (Press -> Stacker) toStacker.DieCutter.fltActualSidewaysPosition
        [7]   // (Press -> Stacker) toStacker.PrintStation[1].fltActualRegisterPosition
        [3].17   // (Press -> Stacker) toStacker.PrintStation[3].blnSideWaysActive
        [8]   // (Press -> Stacker) toStacker.PrintStation[2].fltActualRegisterPosition
        [3].25   // (Press -> Stacker) toStacker.DieCutter.blnDieDrumReferenced
        [3].18   // (Press -> Stacker) toStacker.PrintStation[4].blnSideWaysActive
        [9]   // (Press -> Stacker) toStacker.PrintStation[3].fltActualRegisterPosition
        [3].19   // (Press -> Stacker) toStacker.PrintStation[5].blnSideWaysActive
        [3].20   // (Press -> Stacker) toStacker.PrintStation[6].blnSideWaysActive
        [3].21   // (Press -> Stacker) toStacker.PrintStation[7].blnSideWaysActive
        [3].4   // (Press -> Stacker) toStacker.SheetCountPulseStatus
        [3].7   // (Press -> Stacker) toStacker.DieCutter.blnSpeedChangeActive
        [22]   // (Press -> Stacker) toStacker.Spare1
        [23]   // (Press -> Stacker) toStacker.Spare2
        [3].23   // (LIC -> Stacker) toStacker.ReadyRightAngleForward
        [3].24   // (LIC -> Stacker) toStacker.ReadyRightAngleReverse
        [4]   // (Press -> Stacker) toStacker.DieCutter.uiActualSpeedKpm
        [24]   // Spare
        [25]   // Spare
        [3].0   // (Press -> Stacker) toStacker.RollInPermissive
        [26]   // Spare
        [27]   // Spare
        [28]   // Spare
        [29]   // Spare
        [30]   // Spare
        [31]   // Spare
        [3].2   // (Press -> Stacker) toStacker.VOSReset
        [3].3   // (Press -> Stacker) toStacker.VOSStart
        [21]   // (Interlock -> Stacker) toStacker.CommsStatus
        [1]   // (Press -> Stacker) toStacker.CommandedSpeed
        [0]   // (Press -> Stacker) toStacker.Heartbeat
        [2]   // (Press -> Stacker) toStacker.PressCurrentSpeed
        [3].1   // (Press -> Stacker) toStacker.RunPermissive
        [10]   // (Press -> Stacker) toStacker.PrintStation[4].fltActualRegisterPosition
        [11]   // (Press -> Stacker) toStacker.PrintStation[5].fltActualRegisterPosition
        [12]   // (Press -> Stacker) toStacker.PrintStation[6].fltActualRegisterPosition
        [13]   // (Press -> Stacker) toStacker.PrintStation[7].fltActualRegisterPosition
        [14]   // (Press -> Stacker) toStacker.PrintStation[1].fltActualSidewaysPosition
        [15]   // (Press -> Stacker) toStacker.PrintStation[2].fltActualSidewaysPosition
        [16]   // (Press -> Stacker) toStacker.PrintStation[3].fltActualSidewaysPosition
        [17]   // (Press -> Stacker) toStacker.PrintStation[4].fltActualSidewaysPosition
        [18]   // (Press -> Stacker) toStacker.PrintStation[5].fltActualSidewaysPosition
        [19]   // (Press -> Stacker) toStacker.PrintStation[6].fltActualSidewaysPosition
        [20]   // (Press -> Stacker) toStacker.PrintStation[7].fltActualSidewaysPosition
        [3]   // Bits used: 0-25
        [3].10   // (Press -> Stacker) toStacker.PrintStation[3].blnRegistrationActive
        [3].11   // (Press -> Stacker) toStacker.PrintStation[4].blnRegistrationActive
        [3].12   // (Press -> Stacker) toStacker.PrintStation[5].blnRegistrationActive
        [3].13   // (Press -> Stacker) toStacker.PrintStation[6].blnRegistrationActive
        [3].14   // (Press -> Stacker) toStacker.PrintStation[7].blnRegistrationActive
END_VAR

PROGRAM Fault_Handler_Program   (* main routine ControllerFaultHandlerRoutine, fault routine CheckSpecificFaultRoutine *)
VAR
   CPU_Scanning : BOOL;   // Identifies when the controller is in prescan.Used t to determine if the fault occurred during prescan or normal scan of the logic
   FaultCode : DINT := 20;
   FaultType : DINT := 4;
   MajorFaultRecord : UDT_FaultRecord;
        .TimeLow   // Stores the fault information in the major_fault_record tag. When you enter a tag that is based on a structure, enter the first member of the tag
   MF_ClearRequestEnable : BOOL;   // allow program to clear this class of fault
   MF_Code : DINT;
   MF_Latched : BOOL;   // Goes true when new fault captured
   MF_Msg : STRING;
   MF_T01_C01 : STR_MajorFault := 'Major Fault T01:C01 - Power-up Fault: Power lost and restored in RUN mode. The controller that is powered on is in Run mode.'; {constant}   // The controller that is powered on is in Run mode.
   MF_T01_C16 : STR_MajorFault := 'Major Fault T01:C16 - Power-up Fault: I/O Communications Configuration fault detected.. I/O communication configuration fault detected.'; {constant}   // I/O communication configuration fault detected.
   MF_T01_C60 : STR_MajorFault := 'Major Fault T01:C60 - Power-up Fault: Non-recoverable fault. The controller detected a nonrecoverable major fault. Diagnostic information can be recovered.'; {constant}   // The controller detected a nonrecoverable major fault. Diagnostic information can be recovered.
   MF_T01_C61 : STR_MajorFault := 'Major Fault T01:C61 - Power-up Fault: Non-recoverable fault with saved diagnostic information. The controller detected a nonrecoverable major fault. Diagnostic information can be recovered.'; {constant}   // The controller detected a nonrecoverable major fault. Diagnostic information can be recovered.
   MF_T03_C16 : STR_MajorFault := 'Major Fault T03:C16 - I/O Fault: I/O module connection failed on required module. A required I/O module connection failed.'; {constant}   // A required I/O module connection failed.
   MF_T03_C23 : STR_MajorFault := 'Major Fault T03:C23 - I/O Fault: At least one required connection not established before going into RUN mode. At least one required connection was not established before going to Run mode.'; {constant}   // At least one required connection was not established before going to Run mode.
   MF_T03_C32 : STR_MajorFault := 'Major Fault T03:C32 - I/O Fault: Controller failed to open an I/O connection to a fault-tolerant I/O module because its partner controller is in a Primary state. The controller failed to open an I/O c'; {constant}   // The controller failed to open an I/O connection to a fault-tolerant I/O module because its partner controller is in a Primary state.
   MF_T03_C94 : STR_MajorFault := 'Minor Fault T03:C94 - I/O Fault: Module RPI overlap detected. The current RPI update of an I/O module overlaps with its previous RPI update.'; {constant}   // The current RPI update of an I/O module overlaps with its previous RPI update.
   MF_Timestamp : DINT;   // UTC seconds/millis, optional timestamp
   MF_Type : DINT;
END_VAR

ROUTINE CheckSpecificFaultRoutine   (* ladder *)
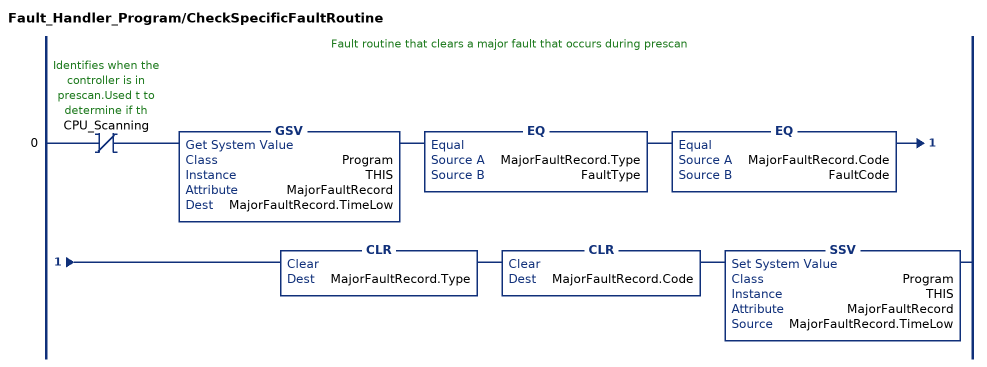
   // Fault routine that clears a major fault that occurs during prescan
   0: XIO(CPU_Scanning)GSV(Program,THIS,MajorFaultRecord,MajorFaultRecord.TimeLow)EQ(MajorFaultRecord.Type,FaultType)EQ(MajorFaultRecord.Code,FaultCode)CLR(MajorFaultRecord.Type)CLR(MajorFaultRecord.Code)SSV(Program,THIS,MajorFaultRecord,MajorFaultRecord.TimeLow);
END_ROUTINE

ROUTINE ControllerFaultHandlerRoutine   (* ladder *)
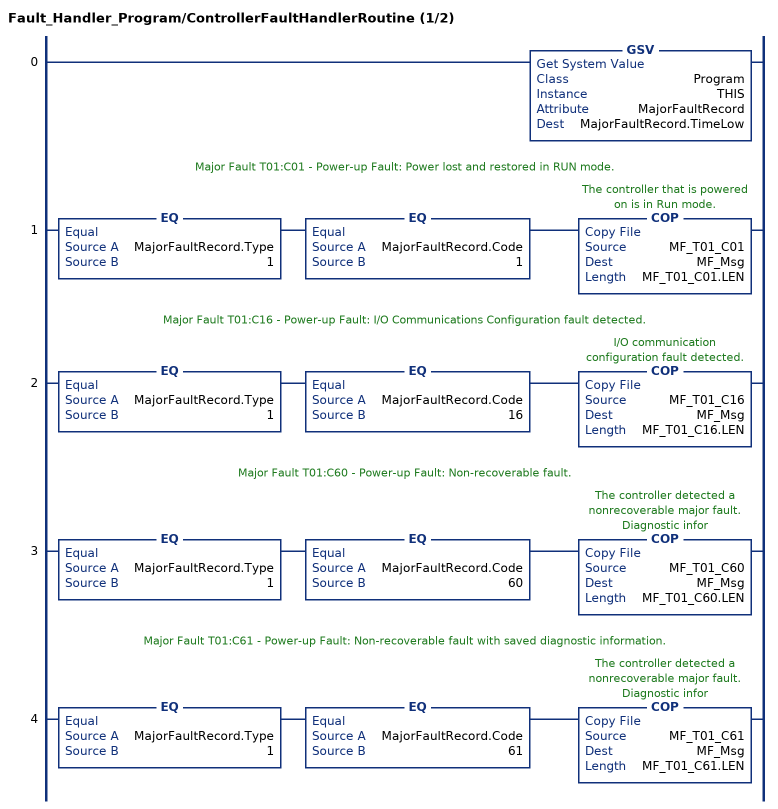
   0: GSV(Program,THIS,MajorFaultRecord,MajorFaultRecord.TimeLow);
   // Major Fault T01:C01 - Power-up Fault: Power lost and restored in RUN mode.
   1: EQ(MajorFaultRecord.Type,1)EQ(MajorFaultRecord.Code,1)COP(MF_T01_C01,MF_Msg,MF_T01_C01.LEN);
   // Major Fault T01:C16 - Power-up Fault: I/O Communications Configuration fault detected.
   2: EQ(MajorFaultRecord.Type,1)EQ(MajorFaultRecord.Code,16)COP(MF_T01_C16,MF_Msg,MF_T01_C16.LEN);
   // Major Fault T01:C60 - Power-up Fault: Non-recoverable fault.
   3: EQ(MajorFaultRecord.Type,1)EQ(MajorFaultRecord.Code,60)COP(MF_T01_C60,MF_Msg,MF_T01_C60.LEN);
   // Major Fault T01:C61 - Power-up Fault: Non-recoverable fault with saved diagnostic information.
   4: EQ(MajorFaultRecord.Type,1)EQ(MajorFaultRecord.Code,61)COP(MF_T01_C61,MF_Msg,MF_T01_C61.LEN);
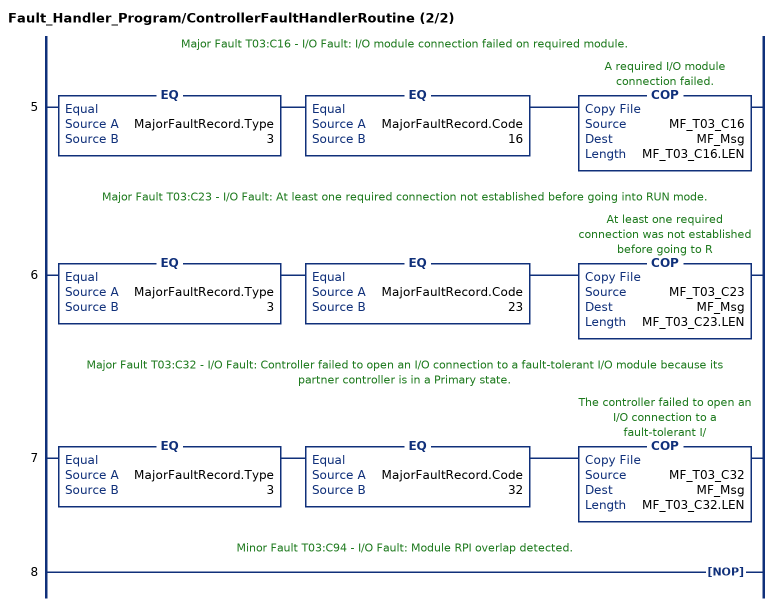
   // Major Fault T03:C16 - I/O Fault: I/O module connection failed on required module.
   5: EQ(MajorFaultRecord.Type,3)EQ(MajorFaultRecord.Code,16)COP(MF_T03_C16,MF_Msg,MF_T03_C16.LEN);
   // Major Fault T03:C23 - I/O Fault: At least one required connection not established before going into RUN mode.
   6: EQ(MajorFaultRecord.Type,3)EQ(MajorFaultRecord.Code,23)COP(MF_T03_C23,MF_Msg,MF_T03_C23.LEN);
   // Major Fault T03:C32 - I/O Fault: Controller failed to open an I/O connection to a fault-tolerant I/O module because its partner controller is in a Primary state.
   7: EQ(MajorFaultRecord.Type,3)EQ(MajorFaultRecord.Code,32)COP(MF_T03_C32,MF_Msg,MF_T03_C32.LEN);
   // Minor Fault T03:C94 - I/O Fault: Module RPI overlap detected.
   8: NOP();
END_ROUTINE
END_PROGRAM

PROGRAM HeartbeatProgram   (* main routine HeartbeatRoutine *)

ROUTINE HeartbeatRoutine   (* ladder *)
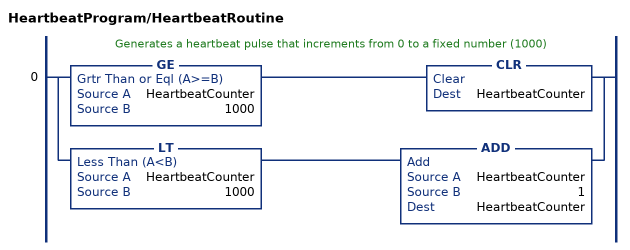
   // Generates a heartbeat pulse that increments from 0 to a fixed number (1000)
   0: [GE(HeartbeatCounter,1000) CLR(HeartbeatCounter) ,LT(HeartbeatCounter,1000) ADD(HeartbeatCounter,1,HeartbeatCounter) ];
END_ROUTINE
END_PROGRAM

PROGRAM MainProgram   (* main routine MainRoutine *)
VAR
   AlwaysTrue : BOOL := 1; {constant}
   Comms : UDT_Comms := (PF.Healthy := 1, PF.Heartbeat := 798, PR.Healthy := 1, PR.Heartbeat := 60636, ST.Healthy := 1, ST.Heartbeat := 60636);
   CommsHealthy : BOOL := 1;   // All machines are communicating
   HWReady : BOOL;   // Machines present and communicating
   InhibitPrefeeder : DINT;
   InhibitPress : DINT;
   InhibitStacker : DINT;
   MajorFaultRec : UDT_FaultRecord;
   MaxScans : DINT := 500; {constant}
   MonitorPFLatency : AOI_Monitor_Comms;   // Calculate Prefeeder Latency characteristics
   MonitorPRLatency : AOI_Monitor_Comms;   // Calculate Press Latency characteristics
   MonitorSTLatency : AOI_Monitor_Comms;   // Calculate Stacker Latency characteristics
   PrefeederHBDetect : AOI_Detect_Heartbeat := (Inp_Heartbeat := 804, Out_Heartbeat_Healthy := 1);
   PressHBDetect : AOI_Detect_Heartbeat := (Inp_Heartbeat := 60636, Out_WD_ACC := 235, Out_WD_EN := 1, Out_Heartbeat_Healthy := 1);
   StackerHBDetect : AOI_Detect_Heartbeat := (Inp_Heartbeat := 60636, Out_WD_ACC := 300, Out_WD_EN := 1, Out_Heartbeat_Healthy := 1);
   StackerLatency_AOI : AOI_Monitor_Comms;
   TaskPeriod_ms : DINT := 10; {constant}   // must match periodic task ms
END_VAR

ROUTINE MainRoutine   (* ladder *)
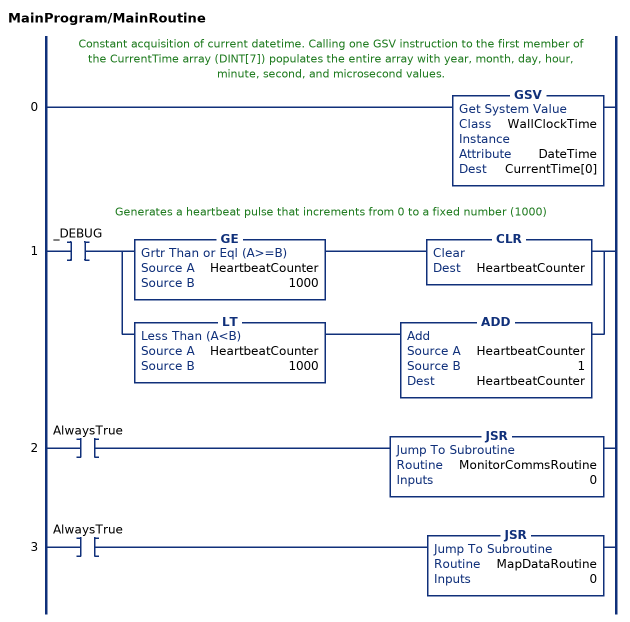
   // Constant acquisition of current datetime. Calling one GSV instruction to the first member of the CurrentTime array (DINT[7]) populates the entire array with year, month, day, hour, minute, second, and microsecond values.
   0: GSV(WallClockTime,,DateTime,CurrentTime[0]);
   // Generates a heartbeat pulse that increments from 0 to a fixed number (1000)
   1: XIC(_DEBUG)[GE(HeartbeatCounter,1000) CLR(HeartbeatCounter) ,LT(HeartbeatCounter,1000) ADD(HeartbeatCounter,1,HeartbeatCounter) ];
   2: XIC(AlwaysTrue)JSR(MonitorCommsRoutine,0);
   3: XIC(AlwaysTrue)JSR(MapDataRoutine,0);
END_ROUTINE

ROUTINE MapDataRoutine   (* structured text *)
   (*
    _____________________________________________________________________________________________
   |                                                    										  |
   |                     DATA MAPPING based on the DINT Mapping Interfaces  					  |
   |_____________________________________________________________________________________________|
   Reference:
   
   	*** Signals ***
   		FromPrefeeder --> Input Message from Prefeeder to Interlock
   		ST1:I.Data 	  --> Input channels from Stacker to Interlock
   		PR1:I.Data 	  --> Input channels from Press to Interlock
   
   		ToPrefeeder2  --> Output Message from Interlock to Prefeeder
   		ST1:O.Data 	  --> Output channels from Interlock to Stacker
   		PR1:O.Data 	  --> Output channels from Interlock to Press
   
   	*** Heartbeats ***
   		Heartbeats are received and sent in two different regions:
   
   			1) region /*--------------- HEARTBEATS IN ------------------*/
   						Heartbeats to Interlock from Machines
   			2) region /*--------------- HEARTBEATS OUT ------------------*/
   						Heartbeat from Interlock to Machines
   
   		The specific mappings are isolated from the main regions and are placed
   		in the respective HEARTBEATS region. For example,
   		PrefeederData.From[3] := FromPrefeeder[3] (heartbeat from the Prefeeder)
   		will be found in the HEARTBEATS IN region and not the PREFEEDER -> INTERLOCK
   		region.
   
   
   	***** CommsStatus ***
   		The CommsStatus DINT has its bits assigned in MainProgram - MonitorCommsRoutine, but
   		the CommsStatus DINT is sent to the machines in this task (MainProgram - MapDataRoutine)
   		in the region:
   
   		region /*--------------- COMMUNICATION STATUS ------------------*/
   *)
   
   
   #region /*--------------- HEARTBEATS IN ------------------*/
   
   PrefeederData.From[3] := FromPrefeeder[3];			//(PreFeeder -> Interlock) Heartbeat
   Comms.PF.Heartbeat	:= FromPrefeeder[3];  					//(Pre-Feeder -> Interlock) FromPrefeeder.Heartbeat DINT
   Comms.PR.Heartbeat 	:= PR1:I.Data[0];						//(Press -> Interlock) fromPress.Heartbeat UINT
   Comms.ST.Heartbeat 	:= ST1:I.Data[0];						//(Stacker -> Interlock) fromStacker.Heartbeat UINT
   
   #endregion
   
   
   
   //#region /*--------------- HEARTBEATS OUT ------------------*/
   
   //#endregion
   
   ////Send Heartbeat to Press FOR TESTING
   //PR1:O.Data[0] := HeartbeatCounter;
   //PR1:O.Data[1] := HeartbeatCounter;
   
   //#region /*--------------- COMMUNICATION STATUS ------------------*/
   //PrefeederData.To[9] := CommsStatus;
   //PR1:O.Data[28] := CommsStatus;
   //ST1:O.Data[23] := CommsStatus;
   //#endregion
   
   #region /*--------------- PREFEEDER -> INTERLOCK ----------------*/
   
   PrefeederData.From[0].0 := FromPrefeeder[0].0;	 	//(PreFeeder -> Interlock) AuxTamperAirRight
   PrefeederData.From[0].1 := FromPrefeeder[0].1;	 	//(PreFeeder -> Interlock) AuxTamperAirLeft
   PrefeederData.From[0].2 := FromPrefeeder[0].2;	 	//(PreFeeder -> Interlock) BackstopInhibit
   PrefeederData.From[0].3 := FromPrefeeder[0].3;	 	//(PreFeeder -> Interlock) CallForStack
   PrefeederData.From[0].4 := FromPrefeeder[0].4;	 	//(PreFeeder -> Interlock) ExtendoUpDown
   PrefeederData.From[0].5 := FromPrefeeder[0].5;	 	//(PreFeeder -> Interlock) EstopFeedbackChannel1
   PrefeederData.From[0].6 := FromPrefeeder[0].6;	 	//(PreFeeder -> Interlock) EstopFeedbackChannel2
   PrefeederData.From[0].7 := FromPrefeeder[0].7;	 	//(PreFeeder -> Interlock) FeedBoardOk
   PrefeederData.From[0].8 := FromPrefeeder[0].8;	 	//(PreFeeder -> Interlock) MachineOpenCloseDisable
   PrefeederData.From[0].9 := FromPrefeeder[0].9;	 	//(PreFeeder -> Interlock) OpenMachineOk
   PrefeederData.From[0].10 := FromPrefeeder[0].10;	//(PreFeeder -> Interlock) ReadyForSetup
   PrefeederData.From[0].11 := FromPrefeeder[0].11;	//(PreFeeder -> Interlock) ReadyToRaise
   PrefeederData.From[0].12 := FromPrefeeder[0].12;	//(PreFeeder -> Interlock) RunEmpty
   PrefeederData.From[0].13 := FromPrefeeder[0].13;	//(PreFeeder -> Interlock) RunForward
   PrefeederData.From[0].14 := FromPrefeeder[0].14;	//(PreFeeder -> Interlock) RunReverse
   PrefeederData.From[0].15 := FromPrefeeder[0].15;	//(PreFeeder -> Interlock) TamperInterrupt
   PrefeederData.From[0].16 := FromPrefeeder[0].16;	//(PreFeeder -> Interlock) Empty
   PrefeederData.From[0].17 := FromPrefeeder[0].17;	//(PreFeeder -> Interlock) FeedInterrupt
   PrefeederData.From[0].18 := FromPrefeeder[0].18;	//(PreFeeder -> Interlock) Spare
   PrefeederData.From[1] := FromPrefeeder[1];			//(PreFeeder -> Interlock) CurrentSpeed
   PrefeederData.From[2] := FromPrefeeder[2];			//(PreFeeder -> Interlock) PatternMaxSpeed
   
   PrefeederData.From[4] := FromPrefeeder[4];			//(PreFeeder -> Interlock) Spare1
   PrefeederData.From[5] := FromPrefeeder[5];			//(PreFeeder -> Interlock) Spare2
   #endregion
   
   #region /*--------------- PRESS -> INTERLOCK --------------------*/
   
   FromPress[0] := PR1:I.Data[0];						//(Press -> Interlock) Hearbeat 	UINT
   FromPress[1] := PR1:I.Data[1];						//(Press -> Interlock) CommandedSpeed	INT
   FromPress[2] := PR1:I.Data[2];						//(Press -> Interlock) CurrentSpeed	INT
   FromPress[3].0 := PR1:I.Data[3].0; 					//(Press -> Interlock) RollInPermissive	BOOL
   FromPress[3].1 := PR1:I.Data[3].1;					//(Press -> Interlock) RunPermissive	BOOL
   FromPress[3].2 := PR1:I.Data[3].2;					//(Press -> Interlock) VOSReset	BOOL
   FromPress[3].3 := PR1:I.Data[3].3;					//(Press -> Interlock) VOSStart	BOOL
   FromPress[3].4 := PR1:I.Data[3].4;					//(Press -> Interlock) SheetCountPulseStatus	BOOL
   FromPress[3].5 := PR1:I.Data[3].5;					//(Press -> Interlock) DieCutter.blnRegistrationActive	BOOL
   FromPress[3].6 := PR1:I.Data[3].6;					//(Press -> Interlock) DieCutter.blnSidewaysActive	BOOL
   FromPress[3].7 := PR1:I.Data[3].7;					//(Press -> Interlock) DieCutter.blnSpeedChangeActive	BOOL
   FromPress[3].8 := PR1:I.Data[3].8;					//(Press -> Interlock) PrintStation[1].blnRegistrationActive	BOOL
   FromPress[3].9 := PR1:I.Data[3].9;					//(Press -> Interlock) PrintStation[2].blnRegistrationActive	BOOL
   FromPress[3].10 := PR1:I.Data[3].10;				//(Press -> Interlock) PrintStation[3].blnRegistrationActive	BOOL
   FromPress[3].11 := PR1:I.Data[3].11;				//(Press -> Interlock) PrintStation[4].blnRegistrationActive	BOOL
   FromPress[3].12 := PR1:I.Data[3].12;				//(Press -> Interlock) PrintStation[5].blnRegistrationActive	BOOL
   FromPress[3].13 := PR1:I.Data[3].13;				//(Press -> Interlock) PrintStation[6].blnRegistrationActive	BOOL
   FromPress[3].14 := PR1:I.Data[3].14;				//(Press -> Interlock) PrintStation[7].blnRegistrationActive	BOOL
   FromPress[3].15 := PR1:I.Data[3].15;				//(Press -> Interlock) PrintStation[8].blnRegistrationActive	BOOL
   FromPress[3].16 := PR1:I.Data[3].16;				//(Press -> Interlock) PrintStation[1].blnSideWaysActive	BOOL
   FromPress[3].17 := PR1:I.Data[3].17;				//(Press -> Interlock) PrintStation[2].blnSideWaysActive	BOOL
   FromPress[3].18 := PR1:I.Data[3].18;				//(Press -> Interlock) PrintStation[3].blnSideWaysActive	BOOL
   FromPress[3].19 := PR1:I.Data[3].19;				//(Press -> Interlock) PrintStation[4].blnSideWaysActive	BOOL
   FromPress[3].20 := PR1:I.Data[3].20;				//(Press -> Interlock) PrintStation[5].blnSideWaysActive	BOOL
   FromPress[3].21 := PR1:I.Data[3].21;				//(Press -> Interlock) PrintStation[6].blnSideWaysActive	BOOL
   FromPress[3].22 := PR1:I.Data[3].22;				//(Press -> Interlock) PrintStation[7].blnSideWaysActive	BOOL
   FromPress[3].23 := PR1:I.Data[3].23;				//(Press -> Interlock) PrintStation[8].blnSideWaysActive	BOOL
   FromPress[3].24 := PR1:I.Data[3].24;				//(Press -> Interlock) DownstreamReady	BOOL
   FromPress[3].25 := PR1:I.Data[3].25;				//(Press -> Interlock) DownstreamReadyRightAngleForward	BOOL
   FromPress[3].26 := PR1:I.Data[3].26;				//(Press -> Interlock) DownstreamReadyRightAngleReverse	BOOL
   FromPress[3].27 := PR1:I.Data[3].27;				//(Press -> Interlock) DieCutter.blnDieDrumReferenced	BOOL
   FromPress[4] := PR1:I.Data[4];						//(Press -> Interlock) DieCutter.uiActualSpeedKpm	INT
   FromPress[5] := PR1:I.Data[5];						//(Press -> Interlock) DieCutter.fltActualRegisterPosition	REAL
   FromPress[6] := PR1:I.Data[6];						//(Press -> Interlock) DieCutter.fltActualSidewaysPosition	REAL
   FromPress[7] := PR1:I.Data[7];						//(Press -> Interlock) PrintStation[1].fltActualRegisterPosition	REAL
   FromPress[8] := PR1:I.Data[8];						//(Press -> Interlock) PrintStation[2].fltActualRegisterPosition	REAL
   FromPress[9] := PR1:I.Data[9];						//(Press -> Interlock) PrintStation[3].fltActualRegisterPosition	REAL
   FromPress[10] := PR1:I.Data[10];					//(Press -> Interlock) PrintStation[4].fltActualRegisterPosition	REAL
   FromPress[11] := PR1:I.Data[11];					//(Press -> Interlock) PrintStation[5].fltActualRegisterPosition	REAL
   FromPress[12] := PR1:I.Data[12];					//(Press -> Interlock) PrintStation[6].fltActualRegisterPosition	REAL
   FromPress[13] := PR1:I.Data[13];					//(Press -> Interlock) PrintStation[7].fltActualRegisterPosition	REAL
   FromPress[14] := PR1:I.Data[14];					//(Press -> Interlock) PrintStation[8].fltActualRegisterPosition	REAL
   FromPress[15] := PR1:I.Data[15];					//(Press -> Interlock) PrintStation[1].fltActualSidewaysPosition	REAL
   FromPress[16] := PR1:I.Data[16];					//(Press -> Interlock) PrintStation[2].fltActualSidewaysPosition	REAL
   FromPress[17] := PR1:I.Data[17];					//(Press -> Interlock) PrintStation[3].fltActualSidewaysPosition	REAL
   FromPress[18] := PR1:I.Data[18];					//(Press -> Interlock) PrintStation[4].fltActualSidewaysPosition	REAL
   FromPress[19] := PR1:I.Data[19];					//(Press -> Interlock) PrintStation[5].fltActualSidewaysPosition	REAL
   FromPress[20] := PR1:I.Data[20];					//(Press -> Interlock) PrintStation[6].fltActualSidewaysPosition	REAL
   FromPress[21] := PR1:I.Data[21];					//(Press -> Interlock) PrintStation[7].fltActualSidewaysPosition	REAL
   FromPress[22] := PR1:I.Data[22];					//(Press -> Interlock) PrintStation[8].fltActualSidewaysPosition	REAL
   FromPress[23] := PR1:I.Data[23];
   FromPress[24] := PR1:I.Data[24];					//(Press -> Interlock) Spare1	DINT
   FromPress[25] := PR1:I.Data[25];					//(Press -> Interlock) Spare2	DINT
   
   
   // ---------------------------------- COPY DINTs to REALs from Press ------------------------------------------
   
   CPS(FromPress[5], FromPress_Copied[0], 31);			//(Press -> Interlock) DieCutter.fltActualRegisterPosition	REAL
   CPS(FromPress[6], FromPress_Copied[1], 31);			//(Press -> Interlock) DieCutter.fltActualSidewaysPosition	REAL
   CPS(FromPress[7], FromPress_Copied[2], 31);			//(Press -> Interlock) PrintStation[1].fltActualRegisterPosition	REAL
   CPS(FromPress[8], FromPress_Copied[3], 31);			//(Press -> Interlock) PrintStation[2].fltActualRegisterPosition	REAL
   CPS(FromPress[9], FromPress_Copied[4], 31);			//(Press -> Interlock) PrintStation[3].fltActualRegisterPosition	REAL
   CPS(FromPress[10], FromPress_Copied[5], 31);		//(Press -> Interlock) PrintStation[4].fltActualRegisterPosition	REAL
   CPS(FromPress[11], FromPress_Copied[6], 31);		//(Press -> Interlock) PrintStation[5].fltActualRegisterPosition	REAL
   CPS(FromPress[12], FromPress_Copied[7], 31);		//(Press -> Interlock) PrintStation[6].fltActualRegisterPosition	REAL
   CPS(FromPress[13], FromPress_Copied[8], 31);		//(Press -> Interlock) PrintStation[7].fltActualRegisterPosition	REAL
   CPS(FromPress[14], FromPress_Copied[9], 31);		//(Press -> Interlock) PrintStation[8].fltActualRegisterPosition	REAL
   CPS(FromPress[15], FromPress_Copied[10], 31);		//(Press -> Interlock) PrintStation[1].fltActualSidewaysPosition	REAL
   CPS(FromPress[16], FromPress_Copied[11], 31);		//(Press -> Interlock) PrintStation[2].fltActualSidewaysPosition	REAL
   CPS(FromPress[17], FromPress_Copied[12], 31);		//(Press -> Interlock) PrintStation[3].fltActualSidewaysPosition	REAL
   CPS(FromPress[18], FromPress_Copied[13], 31);		//(Press -> Interlock) PrintStation[4].fltActualSidewaysPosition	REAL
   CPS(FromPress[19], FromPress_Copied[14], 31);		//(Press -> Interlock) PrintStation[5].fltActualSidewaysPosition	REAL
   CPS(FromPress[20], FromPress_Copied[15], 31);		//(Press -> Interlock) PrintStation[6].fltActualSidewaysPosition	REAL
   CPS(FromPress[21], FromPress_Copied[16], 31);		//(Press -> Interlock) PrintStation[7].fltActualSidewaysPosition	REAL
   CPS(FromPress[22], FromPress_Copied[17], 31);		//(Press -> Interlock) PrintStation[8].fltActualSidewaysPosition	REAL
   // ------------------------------------------------------------------------------------------------------------
   
   
   #endregion
   
   
   #region /*--------------- STACKER -> INTERLOCK ------------------*/
   CPS(FromStacker[0],ToPress[6],31);
   
   FromStacker[0] := ST1:I.Data[0]; 					//(Stacker -> Interlock) Heartbeat	UINT
   FromStacker[1] := ST1:I.Data[1]; 					//(Stacker -> Interlock) CurrentSpeed	INT
   FromStacker[2] := ST1:I.Data[2]; 					//(Stacker -> Interlock) PatternMaxSpeed	INT
   FromStacker[3] := ST1:I.Data[3]; 					//(Stacker -> Interlock) FillPercentage	INT
   FromStacker[4].0 := ST1:I.Data[4].0;				//(Stacker -> Interlock) RunPermissive	BOOL
   FromStacker[4].1 := ST1:I.Data[4].1; 				//(Stacker -> Interlock) FeedRestart	BOOL
   FromStacker[4].2 := ST1:I.Data[4].2; 				//(Stacker -> Interlock) RolledOutStatus	BOOL
   FromStacker[4].3 := ST1:I.Data[4].3; 				//(Stacker -> Interlock) FeedInterruptStatus	BOOL
   FromStacker[4].4 := ST1:I.Data[4].4; 				//(Stacker -> Interlock) DieCutter.blnFast	BOOL
   FromStacker[4].5 := ST1:I.Data[4].5; 				//(Stacker -> Interlock) DieCutter.blnSlow	BOOL
   FromStacker[4].6 := ST1:I.Data[4].6; 				//(Stacker -> Interlock) DieCutter.blnRegisterAdjustRq	BOOL
   FromStacker[4].7 := ST1:I.Data[4].7; 				//(Stacker -> Interlock) DieCutter.blnRegisterStopAdjustRq	BOOL
   FromStacker[4].8 := ST1:I.Data[4].8; 				//(Stacker -> Interlock) DieCutter.blnSidewaysAdjustRq	BOOL
   FromStacker[4].9 := ST1:I.Data[4].9; 				//(Stacker -> Interlock) DieCutter.blnSidewaysStopAdjustRq	BOOL
   FromStacker[4].10 := ST1:I.Data[4].10;				//(Stacker -> Interlock) DieCutter.blnSpeedChangeRq	BOOL
   FromStacker[4].11 := ST1:I.Data[4].11; 				//(Stacker -> Interlock) DieCutter.blnSpeedChangeStopRq	BOOL
   FromStacker[4].12 := ST1:I.Data[4].12;				//(Stacker -> Interlock) PrintStation[1].blnRegisterAdjustRq	BOOL
   FromStacker[4].13 := ST1:I.Data[4].13; 				//(Stacker -> Interlock) PrintStation[2].blnRegisterAdjustRq	BOOL
   FromStacker[4].14 := ST1:I.Data[4].14; 				//(Stacker -> Interlock) PrintStation[3].blnRegisterAdjustRq	BOOL
   FromStacker[4].15 := ST1:I.Data[4].15; 				//(Stacker -> Interlock) PrintStation[4].blnRegisterAdjustRq	BOOL
   FromStacker[4].16 := ST1:I.Data[4].16; 				//(Stacker -> Interlock) PrintStation[5].blnRegisterAdjustRq	BOOL
   FromStacker[4].17 := ST1:I.Data[4].17;				//(Stacker -> Interlock) PrintStation[6].blnRegisterAdjustRq	BOOL
   FromStacker[4].18 := ST1:I.Data[4].18;				//(Stacker -> Interlock) PrintStation[7].blnRegisterAdjustRq	BOOL
   FromStacker[4].19 := ST1:I.Data[4].19;				//(Stacker -> Interlock) PrintStation[8].blnRegisterAdjustRq	BOOL
   FromStacker[4].20 := ST1:I.Data[4].20;				//(Stacker -> Interlock) PrintStation[1].blnSidewaysAdjustRq	BOOL
   FromStacker[4].21 := ST1:I.Data[4].21; 				//(Stacker -> Interlock) PrintStation[2].blnSidewaysAdjustRq	BOOL
   FromStacker[4].22 := ST1:I.Data[4].22;				//(Stacker -> Interlock) PrintStation[3].blnSidewaysAdjustRq	BOOL
   FromStacker[4].23 := ST1:I.Data[4].23; 				//(Stacker -> Interlock) PrintStation[4].blnSidewaysAdjustRq	BOOL
   FromStacker[4].24 := ST1:I.Data[4].24; 				//(Stacker -> Interlock) PrintStation[5].blnSidewaysAdjustRq	BOOL
   FromStacker[4].25 := ST1:I.Data[4].25; 				//(Stacker -> Interlock) PrintStation[6].blnSidewaysAdjustRq	BOOL
   FromStacker[4].26 := ST1:I.Data[4].26;				//(Stacker -> Interlock) PrintStation[7].blnSidewaysAdjustRq	BOOL
   FromStacker[4].27 := ST1:I.Data[4].27;				//(Stacker -> Interlock) PrintStation[8].blnSidewaysAdjustRq	BOOL
   FromStacker[4].28 := ST1:I.Data[4].28; 				//(Stacker -> Interlock) PrintStation[1].blnRegisterStopAdjustRq	BOOL
   FromStacker[4].29 := ST1:I.Data[4].29;				//(Stacker -> Interlock) PrintStation[2].blnRegisterStopAdjustRq	BOOL
   FromStacker[4].30 := ST1:I.Data[4].30; 				//(Stacker -> Interlock) PrintStation[3].blnRegisterStopAdjustRq	BOOL
   FromStacker[4].31 := ST1:I.Data[4].31; 				//(Stacker -> Interlock) PrintStation[4].blnRegisterStopAdjustRq	BOOL
   FromStacker[5].0 := ST1:I.Data[5].0;				//(Stacker -> Interlock) PrintStation[5].blnRegisterStopAdjustRq	BOOL
   FromStacker[5].1 := ST1:I.Data[5].1;				//(Stacker -> Interlock) PrintStation[6].blnRegisterStopAdjustRq	BOOL
   FromStacker[5].2 := ST1:I.Data[5].2;				//(Stacker -> Interlock) PrintStation[7].blnRegisterStopAdjustRq	BOOL
   FromStacker[5].3 := ST1:I.Data[5].3;				//(Stacker -> Interlock) PrintStation[8].blnRegisterStopAdjustRq	BOOL
   FromStacker[5].4 := ST1:I.Data[5].4; 				//(Stacker -> Interlock) PrintStation[1].blnSidewaysStopAdjustRq	BOOL
   FromStacker[5].5 := ST1:I.Data[5].5; 				//(Stacker -> Interlock) PrintStation[2].blnSidewaysStopAdjustRq	BOOL
   FromStacker[5].6 := ST1:I.Data[5].6; 				//(Stacker -> Interlock) PrintStation[3].blnSidewaysStopAdjustRq	BOOL
   FromStacker[5].7 := ST1:I.Data[5].7; 				//(Stacker -> Interlock) PrintStation[4].blnSidewaysStopAdjustRq	BOOL
   FromStacker[5].8 := ST1:I.Data[5].8; 				//(Stacker -> Interlock) PrintStation[5].blnSidewaysStopAdjustRq	BOOL
   FromStacker[5].9 := ST1:I.Data[5].9; 				//(Stacker -> Interlock) PrintStation[6].blnSidewaysStopAdjustRq	BOOL
   FromStacker[5].10 := ST1:I.Data[5].10; 				//(Stacker -> Interlock) PrintStation[7].blnSidewaysStopAdjustRq	BOOL
   FromStacker[5].11 := ST1:I.Data[5].11; 				//(Stacker -> Interlock) PrintStation[8].blnSidewaysStopAdjustRq	BOOL
   FromStacker[6] := ST1:I.Data[6]; 					//(Stacker -> Interlock) DieCutter.uiDesiredSpeedKpm INT
   FromStacker[7] := ST1:I.Data[7]; 					//(Stacker -> Interlock) DieCutter.fltDesiredRegisterAdjust REAL
   FromStacker[8] := ST1:I.Data[8]; 					//(Stacker -> Interlock) PrintStation[1].fltDesiredRegisterAdjust REAL
   FromStacker[9] := ST1:I.Data[9]; 					//(Stacker -> Interlock) PrintStation[2].fltDesiredRegisterAdjust REAL
   FromStacker[10] := ST1:I.Data[10]; 					//(Stacker -> Interlock) PrintStation[3].fltDesiredRegisterAdjust REAL
   FromStacker[11] := ST1:I.Data[11]; 					//(Stacker -> Interlock) PrintStation[4].fltDesiredRegisterAdjust REAL
   FromStacker[12] := ST1:I.Data[12]; 					//(Stacker -> Interlock) PrintStation[5].fltDesiredRegisterAdjust REAL
   FromStacker[13] := ST1:I.Data[13]; 					//(Stacker -> Interlock) PrintStation[6].fltDesiredRegisterAdjust REAL
   FromStacker[14] := ST1:I.Data[14]; 					//(Stacker -> Interlock) PrintStation[7].fltDesiredRegisterAdjust REAL
   FromStacker[15] := ST1:I.Data[15]; 					//(Stacker -> Interlock) PrintStation[8].fltDesiredRegisterAdjust REAL
   FromStacker[16] := ST1:I.Data[16]; 					//(Stacker -> Interlock) DieCutter.fltDesiredSidewaysAdjust REAL
   FromStacker[17] := ST1:I.Data[17]; 					//(Stacker -> Interlock) PrintStation[1].fltDesiredSidewaysAdjust REAL
   FromStacker[18] := ST1:I.Data[18]; 					//(Stacker -> Interlock) PrintStation[2].fltDesiredSidewaysAdjust REAL
   FromStacker[19] := ST1:I.Data[19]; 					//(Stacker -> Interlock) PrintStation[3].fltDesiredSidewaysAdjust REAL
   FromStacker[20] := ST1:I.Data[20]; 					//(Stacker -> Interlock) PrintStation[4].fltDesiredSidewaysAdjust REAL
   FromStacker[21] := ST1:I.Data[21];  				//(Stacker -> Interlock) PrintStation[5].fltDesiredSidewaysAdjust REAL
   FromStacker[22] := ST1:I.Data[22]; 					//(Stacker -> Interlock) PrintStation[6].fltDesiredSidewaysAdjust REAL
   FromStacker[23] := ST1:I.Data[23]; 					//(Stacker -> Interlock) PrintStation[7].fltDesiredSidewaysAdjust REAL
   FromStacker[24] := ST1:I.Data[24]; 					//(Stacker -> Interlock) PrintStation[8].fltDesiredSidewaysAdjust REAL
   FromStacker[25] := ST1:I.Data[25]; 					//(Stacker -> Interlock) PrintStation[8].fltDesiredSidewaysAdjust REAL WRONG
   FromStacker[26] := ST1:I.Data[26]; 					//(Stacker -> Interlock) PrintStation[8].fltDesiredSidewaysAdjust REAL WRONG
   FromStacker[27] := ST1:I.Data[27]; 					//(Stacker -> Interlock) PrintStation[8].fltDesiredSidewaysAdjust REAL WRONG
   FromStacker[28] := ST1:I.Data[28]; 					//(Stacker -> Interlock) PrintStation[8].fltDesiredSidewaysAdjust REAL WRONG
   FromStacker[29] := ST1:I.Data[29]; 					//(Stacker -> Interlock) PrintStation[8].fltDesiredSidewaysAdjust REAL WRONG
   FromStacker[30] := ST1:I.Data[30]; 					//(Stacker -> Interlock) PrintStation[8].fltDesiredSidewaysAdjust REAL WRONG
   
   
   // ---------------------------------- COPY DINTs to REALs from Stacker ------------------------------------------
   
   CPS(ST1:I.Data[7], FromStacker_Copied[0],31);			//(Stacker -> Interlock) DieCutter.fltDesiredRegisterAdjust REAL
   CPS(ST1:I.Data[8], FromStacker_Copied[1],31);			//(Stacker -> Interlock) PrintStation[1].fltDesiredRegisterAdjust REAL
   CPS(ST1:I.Data[9], FromStacker_Copied[2],31);			//(Stacker -> Interlock) PrintStation[2].fltDesiredRegisterAdjust REAL
   CPS(ST1:I.Data[10], FromStacker_Copied[3],31);			//(Stacker -> Interlock) PrintStation[3].fltDesiredRegisterAdjust REAL
   CPS(ST1:I.Data[11], FromStacker_Copied[4],31);			//(Stacker -> Interlock) PrintStation[4].fltDesiredRegisterAdjust REAL
   CPS(ST1:I.Data[12], FromStacker_Copied[5],31);			//(Stacker -> Interlock) PrintStation[5].fltDesiredRegisterAdjust REAL
   CPS(ST1:I.Data[13], FromStacker_Copied[6],31);			//(Stacker -> Interlock) PrintStation[6].fltDesiredRegisterAdjust REAL
   CPS(ST1:I.Data[14], FromStacker_Copied[7],31);			//(Stacker -> Interlock) PrintStation[7].fltDesiredRegisterAdjust REAL
   CPS(ST1:I.Data[15], FromStacker_Copied[8],31);			//(Stacker -> Interlock) PrintStation[8].fltDesiredRegisterAdjust REAL
   CPS(ST1:I.Data[16], FromStacker_Copied[9],31);			//(Stacker -> Interlock) DieCutter.fltDesiredSidewaysAdjust REAL
   CPS(ST1:I.Data[17], FromStacker_Copied[10],31);			//(Stacker -> Interlock) PrintStation[1].fltDesiredSidewaysAdjust REAL
   CPS(ST1:I.Data[18], FromStacker_Copied[11],31);			//(Stacker -> Interlock) PrintStation[2].fltDesiredSidewaysAdjust REAL
   CPS(ST1:I.Data[19], FromStacker_Copied[12],31);			//(Stacker -> Interlock) PrintStation[3].fltDesiredSidewaysAdjust REAL
   CPS(ST1:I.Data[20], FromStacker_Copied[13],31);			//(Stacker -> Interlock) PrintStation[4].fltDesiredSidewaysAdjust REAL
   CPS(ST1:I.Data[21], FromStacker_Copied[14],31);			//(Stacker -> Interlock) PrintStation[5].fltDesiredSidewaysAdjust REAL
   CPS(ST1:I.Data[22], FromStacker_Copied[15],31);			//(Stacker -> Interlock) PrintStation[6].fltDesiredSidewaysAdjust REAL
   CPS(ST1:I.Data[23], FromStacker_Copied[16],31);			//(Stacker -> Interlock) PrintStation[7].fltDesiredSidewaysAdjust REAL
   CPS(ST1:I.Data[24], FromStacker_Copied[17],31);			//(Stacker -> Interlock) PrintStation[8].fltDesiredSidewaysAdjust REAL
   
   // ------------------------------------------------------------------------------------------------------------
   
   #endregion
   
   //Send Heartbeat echo to Prefeeder
   PrefeederData.To[8] := FromPrefeeder[3];			//(PreFeeder -> Interlock) Heartbeat DINT
   
   
   
   
   
   MSG(PrefeederMSG);
   
   #region /*--------------- INTERLOCK -> PREFEEDER ----------------*/
   //ToPrefeeder2[0].0 := PrefeederMSG.To[0].0;
   //ToPrefeeder2[0].1 := PrefeederMSG.To[0].1;
   //ToPrefeeder2[0].2 := PrefeederMSG.To[0].2;
   //ToPrefeeder2[0].3 := PrefeederMSG.To[0].3;
   //ToPrefeeder2[0].4 := PrefeederMSG.To[0].4;
   //ToPrefeeder2[0].5 := PrefeederMSG.To[0].5;
   //ToPrefeeder2[0].6 := PrefeederMSG.To[0].6;
   //ToPrefeeder2[0].7 := PrefeederMSG.To[0].7;
   //ToPrefeeder2[0].8 := PrefeederMSG.To[0].8;
   //ToPrefeeder2[0].9 := PrefeederMSG.To[0].9;
   //ToPrefeeder2[0].10 := PrefeederMSG.To[0].10;
   //ToPrefeeder2[1] := PrefeederMSG.To[1];
   //ToPrefeeder2[2] := PrefeederMSG.To[2];
   //ToPrefeeder2[3] := PrefeederMSG.To[3];
   //ToPrefeeder2[4] := PrefeederMSG.To[4];
   //ToPrefeeder2[5] := PrefeederMSG.To[5];
   //ToPrefeeder2[6] := PrefeederMSG.To[6];
   //ToPrefeeder2[7] := PrefeederMSG.To[7];
   //ToPrefeeder2[8] := PrefeederMSG.To[8];
   //ToPrefeeder2[9] := PrefeederMSG.To[9];
   //ToPrefeeder2[10] := PrefeederMSG.To[10];
   //ToPrefeeder2[11] := PrefeederMSG.To[11];
   #endregion
   
   #region /*--------------- INTERLOCK -> PRESS --------------------*/
   PR1:O.Data[0] := ToPress[0];
   PR1:O.Data[1] := ToPress[1];
   PR1:O.Data[2] := ToPress[2];
   PR1:O.Data[3].0 := ToPress[3].0;
   PR1:O.Data[3].1 := ToPress[3].1;
   PR1:O.Data[3].2 := ToPress[3].2;
   PR1:O.Data[3].3 := ToPress[3].3;
   PR1:O.Data[3].4 := ToPress[3].4;
   PR1:O.Data[3].5 := ToPress[3].5;
   PR1:O.Data[3].6 := ToPress[3].6;
   PR1:O.Data[3].7 := ToPress[3].7;
   PR1:O.Data[3].8 := ToPress[3].8;
   PR1:O.Data[3].9 := ToPress[3].9;
   PR1:O.Data[3].10 := ToPress[3].10;
   PR1:O.Data[3].11 := ToPress[3].11;
   PR1:O.Data[3].12 := ToPress[3].12;
   PR1:O.Data[3].13 := ToPress[3].13;
   PR1:O.Data[3].14 := ToPress[3].14;
   PR1:O.Data[3].15 := ToPress[3].15;
   PR1:O.Data[3].16 := ToPress[3].16;
   PR1:O.Data[3].17 := ToPress[3].17;
   PR1:O.Data[3].18 := ToPress[3].18;
   PR1:O.Data[3].19 := ToPress[3].19;
   PR1:O.Data[3].20 := ToPress[3].20;
   PR1:O.Data[3].21 := ToPress[3].21;
   PR1:O.Data[3].22 := ToPress[3].22;
   PR1:O.Data[3].23 := ToPress[3].23;
   PR1:O.Data[3].24 := ToPress[3].24;
   PR1:O.Data[3].25 := ToPress[3].25;
   PR1:O.Data[3].26 := ToPress[3].26;
   PR1:O.Data[3].27 := ToPress[3].27;
   PR1:O.Data[3].28 := ToPress[3].28;
   PR1:O.Data[3].29 := ToPress[3].29;
   PR1:O.Data[3].30 := ToPress[3].30;
   PR1:O.Data[3].31 := ToPress[3].31;
   PR1:O.Data[4] := ToPress[4];
   PR1:O.Data[5] := ToPress[5];
   PR1:O.Data[6] := ToPress[6];
   PR1:O.Data[7] := ToPress[7];
   PR1:O.Data[8] := ToPress[8];
   PR1:O.Data[9] := ToPress[9];
   PR1:O.Data[10] := ToPress[10];
   PR1:O.Data[11] := ToPress[11];
   PR1:O.Data[12] := ToPress[12];
   PR1:O.Data[13] := ToPress[13];
   PR1:O.Data[14] := ToPress[14];
   PR1:O.Data[15] := ToPress[15];
   PR1:O.Data[16] := ToPress[16];
   PR1:O.Data[17] := ToPress[17];
   PR1:O.Data[18] := ToPress[18];
   PR1:O.Data[19] := ToPress[19];
   PR1:O.Data[20] := ToPress[20];
   PR1:O.Data[21] := ToPress[21];
   PR1:O.Data[22] := ToPress[22];
   PR1:O.Data[23] := ToPress[23];
   PR1:O.Data[24] := ToPress[24];
   PR1:O.Data[25] := ToPress[25];
   PR1:O.Data[26] := ToPress[26];
   PR1:O.Data[27] := ToPress[27];
   //PR1:O.Data[28] := ToPress[28];
   PR1:O.Data[29] := ToPress[29];
   PR1:O.Data[30] := ToPress[30];
   PR1:O.Data[31] := ToPress[31];
   PR1:O.Data[32] := ToPress[32];
   PR1:O.Data[33] := ToPress[33];
   PR1:O.Data[34] := ToPress[34];
   PR1:O.Data[35] := ToPress[35];
   PR1:O.Data[36] := ToPress[36];
   PR1:O.Data[37] := ToPress[37];
   PR1:O.Data[38] := ToPress[38];
   PR1:O.Data[39] := ToPress[39];
   
   #endregion
   
   #region /*--------------- INTERLOCK -> STACKER ------------------*/
   //Send Heartbeat to Stacker
   ST1:O.Data[0] := HeartbeatCounter;
   //CPS(FromPress[0],ToStacker[0],32);
   //ST1:O.Data[0] := ToStacker[0];				//(Press -> Stacker) toStacker.Heartbeat
   ST1:O.Data[1] := ToStacker[1];				//(Press -> Stacker) toStacker.CommandedSpeed
   ST1:O.Data[2] := ToStacker[2];				//(Press -> Stacker) toStacker.PressCurrentSpeed
   ST1:O.Data[3].0 := ToStacker[3].0;			//(Press -> Stacker) toStacker.RollInPermissive
   ST1:O.Data[3].1 := ToStacker[3].1;			//(Press -> Stacker) toStacker.RunPermissive
   ST1:O.Data[3].2 := ToStacker[3].2;			//(Press -> Stacker) toStacker.VOSReset
   ST1:O.Data[3].3 := ToStacker[3].3;			//(Press -> Stacker) toStacker.VOSStart
   ST1:O.Data[3].4 := ToStacker[3].4;			//(Press -> Stacker) toStacker.SheetCountPulseStatus
   ST1:O.Data[3].5 := ToStacker[3].5;			//(Press -> Stacker) toStacker.DieCutter.blnRegistrationActive
   ST1:O.Data[3].6 := ToStacker[3].6;			//(Press -> Stacker) toStacker.DieCutter.blnSidewaysAcitve
   ST1:O.Data[3].7 := ToStacker[3].7;			//(Press -> Stacker) toStacker.DieCutter.blnSpeedChangeActive
   ST1:O.Data[3].8 := ToStacker[3].8;			//(Press -> Stacker) toStacker.PrintStation[1].blnRegistrationActive
   ST1:O.Data[3].9 := ToStacker[3].9;			//(Press -> Stacker) toStacker.PrintStation[2].blnRegistrationActive
   ST1:O.Data[3].10 := ToStacker[3].10;			//(Press -> Stacker) toStacker.PrintStation[3].blnRegistrationActive
   ST1:O.Data[3].11 := ToStacker[3].11;			//(Press -> Stacker) toStacker.PrintStation[4].blnRegistrationActive
   ST1:O.Data[3].12 := ToStacker[3].12;			//(Press -> Stacker) toStacker.PrintStation[5].blnRegistrationActive
   ST1:O.Data[3].13 := ToStacker[3].13;			//(Press -> Stacker) toStacker.PrintStation[6].blnRegistrationActive
   ST1:O.Data[3].14 := ToStacker[3].14;			//(Press -> Stacker) toStacker.PrintStation[7].blnRegistrationActive
   
   
   
   ST1:O.Data[3].15 := ToStacker[3].15;			//(Press -> Stacker) toStacker.PrintStation[1].blnSideWaysActive
   ST1:O.Data[3].16 := ToStacker[3].16;			//(Press -> Stacker) toStacker.PrintStation[2].blnSideWaysActive
   ST1:O.Data[3].17 := ToStacker[3].17;			//(Press -> Stacker) toStacker.PrintStation[3].blnSideWaysActive
   ST1:O.Data[3].18 := ToStacker[3].18;			//(Press -> Stacker) toStacker.PrintStation[4].blnSideWaysActive
   ST1:O.Data[3].19 := ToStacker[3].19;			//(Press -> Stacker) toStacker.PrintStation[5].blnSideWaysActive
   ST1:O.Data[3].20 := ToStacker[3].20;			//(Press -> Stacker) toStacker.PrintStation[6].blnSideWaysActive
   ST1:O.Data[3].21 := ToStacker[3].21;			//(Press -> Stacker) toStacker.PrintStation[7].blnSideWaysActive
   
   
   
   ST1:O.Data[3].22 := ToStacker[3].22;			//(LIC -> Stacker) toStacker.DownstreamReady(StraightThru)
   ST1:O.Data[3].23 := ToStacker[3].23;			//(LIC -> Stacker) toStacker.DownstreamReadyRightAngleForward
   ST1:O.Data[3].24 := ToStacker[3].24;			//(LIC -> Stacker) toStacker.DownstreamReadyRightAngleReverse
   ST1:O.Data[3].25 := ToStacker[3].25;			//(LIC -> Stacker) toStacker.DieCutter.blnDieDrumReferenced
   ST1:O.Data[4] := ToStacker[4];				//(Press -> Stacker) toStacker.DieCutter.uiActualSpeedKpm
   ST1:O.Data[5] := ToStacker[5];				//(Press -> Stacker) toStacker.DieCutter.fltActualRegisterPosition
   ST1:O.Data[6] := ToStacker[6];				//(Press -> Stacker) toStacker.DieCutter.fltActualSidewaysPosition
   ST1:O.Data[7] := ToStacker[7];				//(Press -> Stacker) toStacker.PrintStation[1].fltActualRegisterPosition
   ST1:O.Data[8] := ToStacker[8];				//(Press -> Stacker) toStacker.PrintStation[2].fltActualRegisterPosition
   ST1:O.Data[9] := ToStacker[9];				//(Press -> Stacker) toStacker.PrintStation[3].fltActualRegisterPosition
   ST1:O.Data[10] := ToStacker[10];				//(Press -> Stacker) toStacker.PrintStation[4].fltActualRegisterPosition
   ST1:O.Data[11] := ToStacker[11];				//(Press -> Stacker) toStacker.PrintStation[5].fltActualRegisterPosition
   ST1:O.Data[12] := ToStacker[12];				//(Press -> Stacker) toStacker.PrintStation[6].fltActualRegisterPosition
   ST1:O.Data[13] := ToStacker[13];				//(Press -> Stacker) toStacker.PrintStation[7].fltActualRegisterPosition
   ST1:O.Data[14] := ToStacker[14];				//(Press -> Stacker) toStacker.PrintStation[1].fltActualSidewaysPosition
   ST1:O.Data[15] := ToStacker[15];				//(Press -> Stacker) toStacker.PrintStation[2].fltActualSidewaysPosition
   ST1:O.Data[16] := ToStacker[16];				//(Press -> Stacker) toStacker.PrintStation[3].fltActualSidewaysPosition
   ST1:O.Data[17] := ToStacker[17];				//(Press -> Stacker) toStacker.PrintStation[4].fltActualSidewaysPosition
   ST1:O.Data[18] := ToStacker[18];				//(Press -> Stacker) toStacker.PrintStation[5].fltActualSidewaysPosition
   ST1:O.Data[19] := ToStacker[19];				//(Press -> Stacker) toStacker.PrintStation[6].fltActualSidewaysPosition
   ST1:O.Data[20] := ToStacker[20];				//(Press -> Stacker) toStacker.PrintStation[7].fltActualSidewaysPosition
   
   
   
   ST1:O.Data[21] := ToStacker[21];				//(Interlock -> Stacker) toStacker.CommsStatus
   ST1:O.Data[22] := ToStacker[22];				//(Press -> Stacker) toStacker.Spare1
   //ST1:O.Data[23] := ToStacker[23];				//(Press -> Stacker) toStacker.Spare2
   #endregion
   
   #region PREFEEDER -> PRESS
   //PR1:O.Data[0].0 := FromPrefeeder[0].0; 		//(Pre-Feeder -> Press) FromPrefeeder.AuxTamperAirRight
   //PR1:O.Data[0].1 := FromPrefeeder[0].1; 		//(Pre-Feeder -> Press) FromPrefeeder.AuxTamperAirLeft
   //PR1:O.Data[0].2 := FromPrefeeder[0].2; 		//(Pre-Feeder -> Press) FromPrefeeder.BackstopInhibit
   //PR1:O.Data[0].3 := FromPrefeeder[0].3; 		//(Pre-Feeder -> Floor Conv) FromPrefeeder.CallForStack
   //PR1:O.Data[0].4 := FromPrefeeder[0].4; 		//(Pre-Feeder -> Press) FromPrefeeder.ExtendoUpDown
   //PR1:O.Data[0].5 := FromPrefeeder[0].5;		//(Pre-Feeder -> Press) FromPrefeeder.EstopFeedbackChannel1
   //PR1:O.Data[0].6 := FromPrefeeder[0].6; 		//(Pre-Feeder -> Press) FromPrefeeder.EstopFeedbackChannel2
   //PR1:O.Data[0].7 := FromPrefeeder[0].7; 		//(Pre-Feeder -> Press) FromPrefeeder.FeedBoardOk
   //PR1:O.Data[0].8 := FromPrefeeder[0].8; 		//(Pre-Feeder -> Press) FromPrefeeder.MachineOpenCloseDisable
   //PR1:O.Data[0].9 := FromPrefeeder[0].9; 		//(Pre-Feeder -> Press) FromPrefeeder.OpenMachineOk
   //PR1:O.Data[0].10 := FromPrefeeder[0].10; 		//(Pre-Feeder -> Press) FromPrefeeder.ReadyForSetup
   //PR1:O.Data[0].11 := FromPrefeeder[0].11; 		//(Pre-Feeder -> Press) FromPrefeeder.ReadyToRaise
   //PR1:O.Data[0].12 := FromPrefeeder[0].12; 		//(Pre-Feeder -> Press) FromPrefeeder.RunEmpty
   //PR1:O.Data[0].13 := FromPrefeeder[0].13; 		//(Pre-Feeder -> Floor Conv) FromPrefeeder.RunForward
   //PR1:O.Data[0].14 := FromPrefeeder[0].14; 		//(Pre-Feeder -> Floor Conv) FromPrefeeder.RunReverse
   //PR1:O.Data[0].15 := FromPrefeeder[0].15; 		//(Pre-Feeder -> Press) FromPrefeeder.TamperInterrupt
   //PR1:O.Data[0].16 := FromPrefeeder[0].16; 		//(Pre-Feeder -> Press) FromPrefeeder.Empty
   //PR1:O.Data[0].17 := FromPrefeeder[0].17; 		//(Pre-Feeder -> Press) FromPrefeeder.Spare
   //PR1:O.Data[1] := FromPrefeeder[1]; 			//(Pre-Feeder -> Press) FromPrefeeder.CurrentSpeed INT
   //PR1:O.Data[2] := FromPrefeeder[2]; 			//(Pre-Feeder -> Press) FromPrefeeder.PatternMaxSpeed INT
   //PR1:O.Data[3] := FromPrefeeder[3];  			//(Pre-Feeder -> Press) FromPrefeeder.Heartbeat DINT
   //PR1:O.Data[4] := FromPrefeeder[4]; 			//(Pre-Feeder -> Press) FromPrefeeder.Spare1 DINT
   //PR1:O.Data[5] := FromPrefeeder[5]; 			//(Pre-Feeder -> Press) FromPrefeeder.Spare2 DINT
   #endregion
   
   #region STACKER -> PRESS
   //PR1:O.Data[6] := ST1:I.Data[0]; 				//(Stacker -> Press) fromStacker.Heartbeat UINT
   //PR1:O.Data[7] := ST1:I.Data[1];				//(Stacker -> Press) fromStacker.CurrentSpeed INT
   //PR1:O.Data[8] := ST1:I.Data[2];				//(Stacker -> Press) fromStacker.PatternMaxSpeed INT
   //PR1:O.Data[9] := ST1:I.Data[3];				//(Stacker -> Press) fromStacker.FillPercentage INT
   //PR1:O.Data[10].0 := ST1:I.Data[4].0;			//(Stacker -> Press) fromStacker.RunPermissive
   //PR1:O.Data[10].1 := ST1:I.Data[4].1; 			//(Stacker -> Press) fromStacker.FeedRestart
   //PR1:O.Data[10].2 := ST1:I.Data[4].2; 			//(Stacker -> Press) fromStacker.RolledOutStatus
   PR1:O.Data[10].3 := ST1:I.Data[4].3; 			//(Stacker -> Press) fromStacker.FeedInterruptStatus
   //PR1:O.Data[10].4 := ST1:I.Data[4].4; 			//(Stacker -> Press) fromStacker.DieCutter.blnFast
   //PR1:O.Data[10].5 := ST1:I.Data[4].5; 			//(Stacker -> Press) fromStacker.DieCutter.blnSlow
   //PR1:O.Data[10].6 := ST1:I.Data[4].6; 			//(Stacker -> Press) fromStacker.DieCutter.blnRegisterAdjustRq
   //PR1:O.Data[10].7 := ST1:I.Data[4].7; 			//(Stacker -> Press) fromStacker.DieCutter.blnRegisterStopAdjustRq
   //PR1:O.Data[10].8 := ST1:I.Data[4].8; 			//(Stacker -> Press) fromStacker.DieCutter.blnSidewaysAdjustRq
   //PR1:O.Data[10].9 := ST1:I.Data[4].9; 			//(Stacker -> Press) fromStacker.DieCutter.blnSidewaysStopAdjustRq
   //PR1:O.Data[10].10 := ST1:I.Data[4].10; 		//(Stacker -> Press) fromStacker.DieCutter.blnSpeedChangeRq
   //PR1:O.Data[10].11 := ST1:I.Data[4].11; 		//(Stacker -> Press) fromStacker.DieCutter.blnSpeedChangeStopRq
   //PR1:O.Data[10].12 := ST1:I.Data[4].12; 		//(Stacker -> Press) fromStacker.PrintStation[1].blnRegisterAdjustRq
   //PR1:O.Data[10].13 := ST1:I.Data[4].13; 		//(Stacker -> Press) fromStacker.PrintStation[2].blnRegisterAdjustRq
   //PR1:O.Data[10].14 := ST1:I.Data[4].14; 		//(Stacker -> Press) fromStacker.PrintStation[3].blnRegisterAdjustRq
   //PR1:O.Data[10].15 := ST1:I.Data[4].15;	 	//(Stacker -> Press) fromStacker.PrintStation[4].blnRegisterAdjustRq
   //PR1:O.Data[10].16 := ST1:I.Data[4].16;	 	//(Stacker -> Press) fromStacker.PrintStation[5].blnRegisterAdjustRq
   //PR1:O.Data[10].17 := ST1:I.Data[4].17;	 	//(Stacker -> Press) fromStacker.PrintStation[6].blnRegisterAdjustRq
   //PR1:O.Data[10].18 := ST1:I.Data[4].18;	 	//(Stacker -> Press) fromStacker.PrintStation[7].blnRegisterAdjustRq
   
   
   
   //PR1:O.Data[10].19 := ST1:I.Data[4].19;	 	//(Stacker -> Press) fromStacker.PrintStation[1].blnSidewaysAdjustRq
   //PR1:O.Data[10].20 := ST1:I.Data[4].20;	 	//(Stacker -> Press) fromStacker.PrintStation[2].blnSidewaysAdjustRq
   //PR1:O.Data[10].21 := ST1:I.Data[4].21;	 	//(Stacker -> Press) fromStacker.PrintStation[3].blnSidewaysAdjustRq
   //PR1:O.Data[10].22 := ST1:I.Data[4].22;	 	//(Stacker -> Press) fromStacker.PrintStation[4].blnSidewaysAdjustRq
   //PR1:O.Data[10].23 := ST1:I.Data[4].23;		//(Stacker -> Press) fromStacker.PrintStation[5].blnSidewaysAdjustRq
   //PR1:O.Data[10].24 := ST1:I.Data[4].24; 		//(Stacker -> Press) fromStacker.PrintStation[6].blnSidewaysAdjustRq
   //PR1:O.Data[10].25 := ST1:I.Data[4].25;	 	//(Stacker -> Press) fromStacker.PrintStation[7].blnSidewaysAdjustRq
   
   
   
   //PR1:O.Data[10].26 := ST1:I.Data[4].26;	 	//(Stacker -> Press) fromStacker.PrintStation[1].blnRegisterStopAdjustRq
   //PR1:O.Data[10].27 := ST1:I.Data[4].27;	 	//(Stacker -> Press) fromStacker.PrintStation[2].blnRegisterStopAdjustRq
   //PR1:O.Data[10].28 := ST1:I.Data[4].28;	 	//(Stacker -> Press) fromStacker.PrintStation[3].blnRegisterStopAdjustRq
   //PR1:O.Data[10].29 := ST1:I.Data[4].29;	 	//(Stacker -> Press) fromStacker.PrintStation[4].blnRegisterStopAdjustRq
   //PR1:O.Data[10].30 := ST1:I.Data[4].30;	 	//(Stacker -> Press) fromStacker.PrintStation[5].blnRegisterStopAdjustRq
   //PR1:O.Data[10].31 := ST1:I.Data[4].31;	 	//(Stacker -> Press) fromStacker.PrintStation[6].blnRegisterStopAdjustRq
   //PR1:O.Data[11].0 := ST1:I.Data[5].0; 			//(Stacker -> Press) fromStacker.PrintStation[7].blnRegisterStopAdjustRq
   
   
   
   //PR1:O.Data[11].1 := ST1:I.Data[5].1; 			//(Stacker -> Press) fromStacker.PrintStation[1].blnSidewaysStopAdjustRq
   //PR1:O.Data[11].2 := ST1:I.Data[5].2; 			//(Stacker -> Press) fromStacker.PrintStation[2].blnSidewaysStopAdjustRq
   //PR1:O.Data[11].3 := ST1:I.Data[5].3; 			//(Stacker -> Press) fromStacker.PrintStation[3].blnSidewaysStopAdjustRq
   //PR1:O.Data[11].4 := ST1:I.Data[5].4; 			//(Stacker -> Press) fromStacker.PrintStation[4].blnSidewaysStopAdjustRq
   //PR1:O.Data[11].5 := ST1:I.Data[5].5; 			//(Stacker -> Press) fromStacker.PrintStation[5].blnSidewaysStopAdjustRq
   //PR1:O.Data[11].6 := ST1:I.Data[5].6; 			//(Stacker -> Press) fromStacker.PrintStation[6].blnSidewaysStopAdjustRq
   //PR1:O.Data[11].7 := ST1:I.Data[5].7;			//(Stacker -> Press) fromStacker.PrintStation[7].blnSidewaysStopAdjustRq
   
   
   
   //PR1:O.Data[12] := ST1:I.Data[6]; 				//(Stacker -> Press) fromStacker.DieCutter.uiDesiredSpeedKpm INT
   //PR1:O.Data[13] := ST1:I.Data[7]; 				//(Stacker -> Press) fromStacker.DieCutter.fltDesiredRegisterAdjust REAL
   //PR1:O.Data[14] := ST1:I.Data[8]; 				//(Stacker -> Press) fromStacker.PrintStation[1].fltDesiredRegisterAdjust REAL
   //PR1:O.Data[15] := ST1:I.Data[9]; 				//(Stacker -> Press) fromStacker.PrintStation[2].fltDesiredRegisterAdjust REAL
   //PR1:O.Data[16] := ST1:I.Data[10]; 			//(Stacker -> Press) fromStacker.PrintStation[3].fltDesiredRegisterAdjust REAL
   //PR1:O.Data[17] := ST1:I.Data[11]; 			//(Stacker -> Press) fromStacker.PrintStation[4].fltDesiredRegisterAdjust REAL
   //PR1:O.Data[18] := ST1:I.Data[12]; 			//(Stacker -> Press) fromStacker.PrintStation[5].fltDesiredRegisterAdjust REAL
   //PR1:O.Data[19] := ST1:I.Data[13]; 			//(Stacker -> Press) fromStacker.PrintStation[6].fltDesiredRegisterAdjust REAL
   //PR1:O.Data[20] := ST1:I.Data[14]; 			//(Stacker -> Press) fromStacker.PrintStation[7].fltDesiredRegisterAdjust REAL
   
   
   //PR1:O.Data[21] := ST1:I.Data[15]; 			//(Stacker -> Press) fromStacker.DieCutter.fltDesiredSidewaysAdjust REAL
   //PR1:O.Data[22] := ST1:I.Data[16]; 			//(Stacker -> Press) fromStacker.PrintStation[1].fltDesiredSidewaysAdjust REAL
   //PR1:O.Data[23] := ST1:I.Data[17]; 			//(Stacker -> Press) fromStacker.PrintStation[2].fltDesiredSidewaysAdjust REAL
   //PR1:O.Data[24] := ST1:I.Data[18]; 			//(Stacker -> Press) fromStacker.PrintStation[3].fltDesiredSidewaysAdjust REAL
   //PR1:O.Data[25] := ST1:I.Data[19]; 			//(Stacker -> Press) fromStacker.PrintStation[4].fltDesiredSidewaysAdjust REAL
   //PR1:O.Data[26] := ST1:I.Data[20]; 			//(Stacker -> Press) fromStacker.PrintStation[5].fltDesiredSidewaysAdjust REAL
   //PR1:O.Data[27] := ST1:I.Data[21]; 			//(Stacker -> Press) fromStacker.PrintStation[6].fltDesiredSidewaysAdjust REAL
   //PR1:O.Data[28] := ST1:I.Data[22]; 			//(Stacker -> Press) fromStacker.PrintStation[7].fltDesiredSidewaysAdjust REAL
   #endregion
   
   #region PREFEEDER -> INTERLOCK -> PRESS
   //PR1:O.Data[0].0 := PrefeederMSG.To[0].0; 		//(Pre-Feeder -> Press) FromPrefeeder.AuxTamperAirRight
   //PR1:O.Data[0].1 := PrefeederMSG.To[0].1; 		//(Pre-Feeder -> Press) FromPrefeeder.AuxTamperAirLeft
   //PR1:O.Data[0].2 := PrefeederMSG.To[0].2; 		//(Pre-Feeder -> Press) FromPrefeeder.BackstopInhibit
   //PR1:O.Data[0].3 := PrefeederMSG.To[0].3; 		//(Pre-Feeder -> Floor Conv) FromPrefeeder.CallForStack
   //PR1:O.Data[0].4 := PrefeederMSG.To[0].4; 		//(Pre-Feeder -> Press) FromPrefeeder.ExtendoUpDown
   //PR1:O.Data[0].5 := PrefeederMSG.To[0].5;		//(Pre-Feeder -> Press) FromPrefeeder.EstopFeedbackChannel1
   //PR1:O.Data[0].6 := PrefeederMSG.To[0].6; 		//(Pre-Feeder -> Press) FromPrefeeder.EstopFeedbackChannel2
   //PR1:O.Data[0].7 := PrefeederMSG.To[0].7; 		//(Pre-Feeder -> Press) FromPrefeeder.FeedBoardOk
   //PR1:O.Data[0].8 := PrefeederMSG.To[0].8; 		//(Pre-Feeder -> Press) FromPrefeeder.MachineOpenCloseDisable
   //PR1:O.Data[0].9 := PrefeederMSG.To[0].9; 		//(Pre-Feeder -> Press) FromPrefeeder.OpenMachineOk
   //PR1:O.Data[0].10 := PrefeederMSG.To[0].10; 	//(Pre-Feeder -> Press) FromPrefeeder.ReadyForSetup
   //PR1:O.Data[0].11 := PrefeederMSG.To[0].11; 	//(Pre-Feeder -> Press) FromPrefeeder.ReadyToRaise
   //PR1:O.Data[0].12 := PrefeederMSG.To[0].12; 	//(Pre-Feeder -> Press) FromPrefeeder.RunEmpty
   //PR1:O.Data[0].13 := PrefeederMSG.To[0].13; 	//(Pre-Feeder -> Floor Conv) FromPrefeeder.RunForward
   //PR1:O.Data[0].14 := PrefeederMSG.To[0].14; 	//(Pre-Feeder -> Floor Conv) FromPrefeeder.RunReverse
   //PR1:O.Data[0].15 := PrefeederMSG.To[0].15; 	//(Pre-Feeder -> Press) FromPrefeeder.TamperInterrupt
   //PR1:O.Data[0].16 := PrefeederMSG.To[0].16; 	//(Pre-Feeder -> Press) FromPrefeeder.Empty
   //PR1:O.Data[0].17 := PrefeederMSG.To[0].17; 	//(Pre-Feeder -> Press) FromPrefeeder.Spare
   //PR1:O.Data[1] := PrefeederMSG.To[1]; 			//(Pre-Feeder -> Press) FromPrefeeder.CurrentSpeed INT
   //PR1:O.Data[2] := PrefeederMSG.To[2]; 			//(Pre-Feeder -> Press) FromPrefeeder.PatternMaxSpeed INT
   //PR1:O.Data[3] := PrefeederMSG.To[3];  		//(Pre-Feeder -> Press) FromPrefeeder.Heartbeat DINT
   //PR1:O.Data[4] := PrefeederMSG.To[4]; 			//(Pre-Feeder -> Press) FromPrefeeder.Spare1 DINT
   //PR1:O.Data[5] := PrefeederMSG.To[5]; 			//(Pre-Feeder -> Press) FromPrefeeder.Spare2 DINT
   #endregion
   
   #region STACKER -> INTERLOCK -> PRESS
   //PR1:O.Data[6] := FromStacker[0]; 				//(Stacker -> Press) fromStacker.Heartbeat UINT
   //PR1:O.Data[7] := FromStacker[1]; 				//(Stacker -> Press) fromStacker.CurrentSpeed INT
   //PR1:O.Data[8] := FromStacker[2]; 				//(Stacker -> Press) fromStacker.PatternMaxSpeed INT
   //PR1:O.Data[9] := FromStacker[3]; 				//(Stacker -> Press) fromStacker.FillPercentage INT
   //PR1:O.Data[10].0 := FromStacker[4].0;			//(Stacker -> Press) fromStacker.RunPermissive
   //PR1:O.Data[10].1 := FromStacker[4].1; 		//(Stacker -> Press) fromStacker.FeedRestart
   //PR1:O.Data[10].2 := FromStacker[4].2; 		//(Stacker -> Press) fromStacker.RolledOutStatus
   //PR1:O.Data[10].3 := FromStacker[4].3; 		//(Stacker -> Press) fromStacker.FeedInterruptStatus
   //PR1:O.Data[10].4 := FromStacker[4].4; 		//(Stacker -> Press) fromStacker.DieCutter.blnFast
   //PR1:O.Data[10].5 := FromStacker[4].5; 		//(Stacker -> Press) fromStacker.DieCutter.blnSlow
   //PR1:O.Data[10].6 := FromStacker[4].6; 		//(Stacker -> Press) fromStacker.DieCutter.blnRegisterAdjustRq
   //PR1:O.Data[10].7 := FromStacker[4].7; 		//(Stacker -> Press) fromStacker.DieCutter.blnRegisterStopAdjustRq
   //PR1:O.Data[10].8 := FromStacker[4].8; 		//(Stacker -> Press) fromStacker.DieCutter.blnSidewaysAdjustRq
   //PR1:O.Data[10].9 := FromStacker[4].9; 		//(Stacker -> Press) fromStacker.DieCutter.blnSidewaysStopAdjustRq
   //PR1:O.Data[10].10 := FromStacker[4].10; 		//(Stacker -> Press) fromStacker.DieCutter.blnSpeedChangeRq
   //PR1:O.Data[10].11 := FromStacker[4].11; 		//(Stacker -> Press) fromStacker.DieCutter.blnSpeedChangeStopRq
   //PR1:O.Data[10].12 := FromStacker[4].12; 		//(Stacker -> Press) fromStacker.PrintStation[1].blnRegisterAdjustRq
   //PR1:O.Data[10].13 := FromStacker[4].13; 		//(Stacker -> Press) fromStacker.PrintStation[2].blnRegisterAdjustRq
   //PR1:O.Data[10].14 := FromStacker[4].14; 		//(Stacker -> Press) fromStacker.PrintStation[3].blnRegisterAdjustRq
   //PR1:O.Data[10].15 := FromStacker[4].15; 		//(Stacker -> Press) fromStacker.PrintStation[4].blnRegisterAdjustRq
   //PR1:O.Data[10].16 := FromStacker[4].16; 		//(Stacker -> Press) fromStacker.PrintStation[5].blnRegisterAdjustRq
   //PR1:O.Data[10].17 := FromStacker[4].17; 		//(Stacker -> Press) fromStacker.PrintStation[6].blnRegisterAdjustRq
   //PR1:O.Data[10].18 := FromStacker[4].18; 		//(Stacker -> Press) fromStacker.PrintStation[7].blnRegisterAdjustRq
   
   
   
   //PR1:O.Data[10].19 := FromStacker[4].19; 		//(Stacker -> Press) fromStacker.PrintStation[1].blnSidewaysAdjustRq
   //PR1:O.Data[10].20 := FromStacker[4].20; 		//(Stacker -> Press) fromStacker.PrintStation[2].blnSidewaysAdjustRq
   //PR1:O.Data[10].21 := FromStacker[4].21; 		//(Stacker -> Press) fromStacker.PrintStation[3].blnSidewaysAdjustRq
   //PR1:O.Data[10].22 := FromStacker[4].22; 		//(Stacker -> Press) fromStacker.PrintStation[4].blnSidewaysAdjustRq
   //PR1:O.Data[10].23 := FromStacker[4].23; 		//(Stacker -> Press) fromStacker.PrintStation[5].blnSidewaysAdjustRq
   //PR1:O.Data[10].24 := FromStacker[4].24; 		//(Stacker -> Press) fromStacker.PrintStation[6].blnSidewaysAdjustRq
   //PR1:O.Data[10].25 := FromStacker[4].25; 		//(Stacker -> Press) fromStacker.PrintStation[7].blnSidewaysAdjustRq
   
   
   
   //PR1:O.Data[10].26 := FromStacker[4].26; 		//(Stacker -> Press) fromStacker.PrintStation[1].blnRegisterStopAdjustRq
   //PR1:O.Data[10].27 := FromStacker[4].27; 		//(Stacker -> Press) fromStacker.PrintStation[2].blnRegisterStopAdjustRq
   //PR1:O.Data[10].28 := FromStacker[4].28; 		//(Stacker -> Press) fromStacker.PrintStation[3].blnRegisterStopAdjustRq
   //PR1:O.Data[10].29 := FromStacker[4].29; 		//(Stacker -> Press) fromStacker.PrintStation[4].blnRegisterStopAdjustRq
   //PR1:O.Data[10].30 := FromStacker[4].30; 		//(Stacker -> Press) fromStacker.PrintStation[5].blnRegisterStopAdjustRq
   //PR1:O.Data[10].31 := FromStacker[4].31; 		//(Stacker -> Press) fromStacker.PrintStation[6].blnRegisterStopAdjustRq
   //PR1:O.Data[11].0 := FromStacker[5].0; 		//(Stacker -> Press) fromStacker.PrintStation[7].blnRegisterStopAdjustRq
   
   
   
   //PR1:O.Data[11].1 := FromStacker[5].1; 		//(Stacker -> Press) fromStacker.PrintStation[1].blnSidewaysStopAdjustRq
   //PR1:O.Data[11].2 := FromStacker[5].2; 		//(Stacker -> Press) fromStacker.PrintStation[2].blnSidewaysStopAdjustRq
   //PR1:O.Data[11].3 := FromStacker[5].3; 		//(Stacker -> Press) fromStacker.PrintStation[3].blnSidewaysStopAdjustRq
   //PR1:O.Data[11].4 := FromStacker[5].4; 		//(Stacker -> Press) fromStacker.PrintStation[4].blnSidewaysStopAdjustRq
   //PR1:O.Data[11].5 := FromStacker[5].5; 		//(Stacker -> Press) fromStacker.PrintStation[5].blnSidewaysStopAdjustRq
   //PR1:O.Data[11].6 := FromStacker[5].6; 		//(Stacker -> Press) fromStacker.PrintStation[6].blnSidewaysStopAdjustRq
   //PR1:O.Data[11].7 := FromStacker[5].7; 		//(Stacker -> Press) fromStacker.PrintStation[7].blnSidewaysStopAdjustRq
   
   
   
   //PR1:O.Data[12] := FromStacker[6]; 			//(Stacker -> Press) fromStacker.DieCutter.uiDesiredSpeedKpm INT
   //PR1:O.Data[13] := FromStacker[7]; 			//(Stacker -> Press) fromStacker.DieCutter.fltDesiredRegisterAdjust REAL
   //PR1:O.Data[14] := FromStacker[8]; 			//(Stacker -> Press) fromStacker.PrintStation[1].fltDesiredRegisterAdjust REAL
   //PR1:O.Data[15] := FromStacker[9]; 			//(Stacker -> Press) fromStacker.PrintStation[2].fltDesiredRegisterAdjust REAL
   //PR1:O.Data[16] := FromStacker[10]; 			//(Stacker -> Press) fromStacker.PrintStation[3].fltDesiredRegisterAdjust REAL
   //PR1:O.Data[17] := FromStacker[11]; 			//(Stacker -> Press) fromStacker.PrintStation[4].fltDesiredRegisterAdjust REAL
   //PR1:O.Data[18] := FromStacker[12]; 			//(Stacker -> Press) fromStacker.PrintStation[5].fltDesiredRegisterAdjust REAL
   //PR1:O.Data[19] := FromStacker[13]; 			//(Stacker -> Press) fromStacker.PrintStation[6].fltDesiredRegisterAdjust REAL
   //PR1:O.Data[20] := FromStacker[14]; 			//(Stacker -> Press) fromStacker.PrintStation[7].fltDesiredRegisterAdjust REAL
   
   
   
   //PR1:O.Data[21] := FromStacker[15]; 			//(Stacker -> Press) fromStacker.DieCutter.fltDesiredSidewaysAdjust REAL
